C03628=1105.087,205.699,431.695,178.828,14.143,151.207
C03629=1105.092,205.948,431.670,178.832,14.142,151.206
C03630=1105.098,206.197,431.646,178.836,14.141,151.205
C03631=1105.103,206.446,431.621,178.840,14.139,151.203
C03632=1105.109,206.694,431.597,178.845,14.138,151.202
C03633=1105.115,206.943,431.573,178.848,14.136,151.201
C03634=1105.121,207.191,431.548,178.853,14.136,151.200
C03635=1105.126,207.440,431.524,178.857,14.134,151.198
C03636=1105.132,207.689,431.499,178.861,14.133,151.197
C03637=1105.156,208.685,431.402,178.887,14.133,151.191
C03638=1105.163,209.052,431.365,178.893,14.132,151.190
C03639=1105.171,209.419,431.330,178.899,14.131,151.188
C03640=1105.181,209.786,431.293,178.904,14.131,151.187
C03641=1105.189,210.152,431.257,178.911,14.131,151.186
C03642=1105.195,210.402,431.232,178.914,14.129,151.185
C03643=1105.200,210.650,431.208,178.918,14.129,151.184
C03644=1105.206,210.899,431.183,178.922,14.129,151.183
C03645=1105.211,211.147,431.159,178.926,14.129,151.182
C03646=1105.217,211.397,431.134,178.930,14.128,151.181
C03647=1105.223,211.645,431.109,178.934,14.127,151.180
C03648=1105.228,211.893,431.085,178.938,14.127,151.179
C03649=1105.234,212.143,431.060,178.942,14.126,151.178
C03650=1105.240,212.390,431.035,178.946,14.126,151.177
C03651=1105.246,212.640,431.010,178.949,14.125,151.176
C03652=1105.251,212.888,430.986,178.953,14.125,151.175
C03653=1105.256,213.137,430.960,178.958,14.125,151.174
C03654=1105.262,213.386,430.936,178.961,14.125,151.173
C03655=1105.268,213.635,430.911,178.966,14.124,151.172
C03656=1105.273,213.883,430.886,178.969,14.123,151.171
C03657=1105.279,214.132,430.861,178.973,14.123,151.170
C03658=1105.285,214.381,430.836,178.977,14.123,151.169
C03659=1105.291,214.629,430.812,178.981,14.122,151.168
C03660=1105.296,214.879,430.786,178.985,14.122,151.167
C03661=1105.302,215.127,430.761,178.989,14.122,151.166
C03662=1105.308,215.376,430.737,178.993,14.121,151.165
C03663=1105.313,215.624,430.712,178.997,14.120,151.164
C03664=1105.319,215.873,430.687,179.001,14.120,151.163
C03665=1105.325,216.121,430.662,179.005,14.120,151.162
C03666=1105.330,216.371,430.637,179.009,14.119,151.161
C03667=1105.335,216.619,430.612,179.012,14.119,151.160
C03668=1105.341,216.868,430.587,179.017,14.118,151.159
C03669=1105.348,217.117,430.562,179.020,14.118,151.158
C03670=1105.352,217.365,430.536,179.025,14.118,151.157
C03671=1105.358,217.614,430.512,179.029,14.118,151.156
C03672=1105.364,217.862,430.487,179.033,14.117,151.155
C03673=1105.370,218.111,430.461,179.036,14.116,151.154
C03674=1105.375,218.361,430.436,179.040,14.116,151.153
C03675=1105.381,218.608,430.411,179.044,14.116,151.152
C03676=1105.387,218.857,430.386,179.048,14.115,151.151
C03677=1105.392,219.106,430.362,179.052,14.115,151.150
C03678=1105.398,219.355,430.336,179.056,14.115,151.149
C03679=1105.404,219.603,430.310,179.060,14.114,151.148
C03680=1105.409,219.852,430.286,179.064,14.114,151.147
C03681=1105.415,220.101,430.260,179.068,14.113,151.146
C03682=1105.421,220.350,430.235,179.072,14.113,151.145
C03683=1105.427,220.598,430.210,179.076,14.113,151.144
C03684=1105.433,220.847,430.185,179.080,14.112,151.143
C03685=1105.438,221.096,430.159,179.083,14.112,151.142
C03686=1105.444,221.344,430.134,179.087,14.111,151.141
C03687=1105.450,221.592,430.109,179.092,14.111,151.140
C03688=1105.455,221.841,430.083,179.096,14.111,151.139
C03689=1105.461,222.089,430.058,179.100,14.110,151.138
C03690=1105.470,222.460,430.020,179.105,14.110,151.137
C03691=1105.477,222.831,429.983,179.111,14.109,151.135
C03692=1105.486,223.201,429.944,179.117,14.108,151.134
C03693=1105.494,223.571,429.907,179.123,14.108,151.133
C03694=1105.501,223.820,429.881,179.127,14.108,151.132
C03695=1105.506,224.068,429.856,179.131,14.107,151.131
C03696=1105.512,224.316,429.831,179.134,14.107,151.130
C03697=1105.517,224.565,429.805,179.139,14.107,151.129
C03698=1105.523,224.814,429.779,179.143,14.107,151.128
C03699=1105.528,225.062,429.754,179.147,14.106,151.127
C03700=1105.534,225.311,429.728,179.151,14.106,151.126
C03701=1105.540,225.560,429.702,179.155,14.106,151.125
C03702=1105.545,225.808,429.677,179.159,14.106,151.124
C03703=1105.551,226.057,429.652,179.162,14.105,151.123
C03704=1105.556,226.306,429.626,179.166,14.104,151.122
C03705=1105.563,226.555,429.600,179.170,14.104,151.121
C03706=1105.568,226.804,429.574,179.174,14.104,151.120
C03707=1105.574,227.052,429.549,179.178,14.104,151.119
C03708=1105.579,227.301,429.523,179.182,14.103,151.118
C03709=1105.585,227.549,429.498,179.186,14.103,151.117
C03710=1105.591,227.798,429.472,179.191,14.103,151.116
C03711=1105.596,228.047,429.447,179.194,14.102,151.115
C03712=1105.602,228.295,429.421,179.198,14.102,151.114
C03713=1105.608,228.544,429.395,179.202,14.102,151.113
C03714=1105.614,228.792,429.369,179.206,14.102,151.112
C03715=1105.619,229.041,429.343,179.210,14.101,151.111
C03716=1105.625,229.290,429.317,179.214,14.101,151.110
C03717=1105.631,229.538,429.292,179.218,14.101,151.109
C03718=1105.636,229.787,429.266,179.222,14.101,151.108
C03719=1105.642,230.035,429.240,179.226,14.100,151.107
C03720=1105.648,230.284,429.215,179.229,14.100,151.107
C03721=1105.654,230.533,429.188,179.234,14.099,151.105
C03722=1105.659,230.782,429.162,179.237,14.099,151.105
C03723=1105.665,231.030,429.137,179.241,14.099,151.104
C03724=1105.670,231.278,429.111,179.246,14.099,151.103
C03725=1105.676,231.527,429.084,179.250,14.099,151.102
C03726=1105.682,231.776,429.058,179.254,14.098,151.101
C03727=1105.688,232.024,429.033,179.258,14.098,151.100
C03728=1105.693,232.273,429.006,179.262,14.098,151.099
C03729=1105.699,232.522,428.981,179.266,14.098,151.098
C03730=1105.704,232.771,428.955,179.269,14.097,151.097
C03731=1105.710,233.018,428.928,179.273,14.097,151.096
C03732=1105.716,233.267,428.903,179.277,14.097,151.095
C03733=1105.722,233.515,428.876,179.281,14.096,151.094
C03734=1105.727,233.764,428.850,179.285,14.096,151.093
C03735=1105.733,234.013,428.825,179.289,14.096,151.092
C03736=1105.738,234.262,428.798,179.293,14.096,151.091
C03737=1105.744,234.510,428.773,179.297,14.096,151.090
C03738=1105.750,234.759,428.746,179.301,14.096,151.089
C03739=1105.756,235.008,428.720,179.305,14.096,151.089
C03740=1105.762,235.256,428.693,179.309,14.095,151.087
C03741=1105.766,235.504,428.668,179.313,14.095,151.087
C03742=1105.775,235.867,428.629,179.319,14.094,151.085
C03743=1105.783,236.228,428.591,179.324,14.094,151.084
C03744=1105.791,236.590,428.552,179.330,14.094,151.083
C03745=1105.799,236.952,428.514,179.336,14.094,151.081
C03746=1105.805,237.201,428.488,179.340,14.094,151.080
C03747=1105.810,237.449,428.461,179.344,14.093,151.079
C03748=1105.816,237.698,428.436,179.348,14.093,151.078
C03749=1105.822,237.946,428.409,179.351,14.093,151.077
C03750=1105.828,238.194,428.383,179.355,14.092,151.076
C03751=1105.834,238.443,428.357,179.359,14.092,151.075
C03752=1105.839,238.692,428.330,179.363,14.092,151.075
C03753=1105.845,238.940,428.304,179.367,14.092,151.074
C03754=1105.851,239.189,428.278,179.371,14.092,151.073
C03755=1105.856,239.437,428.251,179.375,14.092,151.072
C03756=1105.862,239.686,428.224,179.379,14.091,151.071
C03757=1105.868,239.935,428.198,179.383,14.091,151.070
C03758=1105.874,240.183,428.172,179.387,14.091,151.069
C03759=1105.879,240.432,428.145,179.391,14.091,151.068
C03760=1105.884,240.680,428.118,179.395,14.091,151.067
C03761=1105.890,240.929,428.092,179.399,14.091,151.066
C03762=1105.896,241.178,428.065,179.403,14.091,151.065
C03763=1105.902,241.426,428.038,179.407,14.090,151.064
C03764=1105.908,241.675,428.012,179.411,14.090,151.063
C03765=1105.913,241.923,427.985,179.415,14.090,151.062
C03766=1105.919,242.172,427.958,179.419,14.090,151.061
C03767=1105.925,242.420,427.932,179.423,14.090,151.060
C03768=1105.931,242.669,427.906,179.427,14.090,151.060
C03769=1105.936,242.917,427.879,179.431,14.090,151.059
C03770=1105.942,243.166,427.853,179.435,14.090,151.058
C03771=1105.947,243.414,427.825,179.439,14.090,151.057
C03772=1105.953,243.663,427.799,179.443,14.090,151.056
C03773=1105.959,243.911,427.772,179.446,14.089,151.055
C03774=1105.964,244.159,427.745,179.450,14.089,151.054
C03775=1105.970,244.409,427.718,179.454,14.089,151.053
C03776=1105.976,244.657,427.691,179.458,14.089,151.052
C03777=1105.982,244.905,427.664,179.462,14.089,151.051
C03778=1105.987,245.154,427.638,179.466,14.089,151.050
C03779=1105.992,245.402,427.611,179.470,14.088,151.049
C03780=1105.998,245.651,427.584,179.474,14.088,151.049
C03781=1106.004,245.899,427.557,179.478,14.088,151.048
C03782=1106.010,246.148,427.531,179.482,14.088,151.047
C03783=1106.015,246.396,427.503,179.486,14.088,151.046
C03784=1106.021,246.645,427.476,179.490,14.088,151.045
C03785=1106.027,246.894,427.450,179.494,14.088,151.044
C03786=1106.032,247.142,427.422,179.498,14.088,151.043
C03787=1106.038,247.391,427.396,179.501,14.088,151.042
C03788=1106.043,247.639,427.369,179.505,14.088,151.041
C03789=1106.049,247.888,427.342,179.510,14.087,151.040
C03790=1106.055,248.135,427.315,179.513,14.087,151.039
C03791=1106.060,248.384,427.288,179.517,14.087,151.039
C03792=1106.066,248.633,427.260,179.521,14.087,151.038
C03793=1106.072,248.882,427.234,179.525,14.087,151.037
C03794=1106.079,249.237,427.195,179.531,14.088,151.036
C03795=1106.087,249.591,427.156,179.537,14.087,151.034
C03796=1106.095,249.947,427.117,179.542,14.087,151.033
C03797=1106.104,250.302,427.079,179.548,14.088,151.032
C03798=1106.109,250.550,427.051,179.552,14.088,151.031
C03799=1106.115,250.799,427.024,179.556,14.088,151.030
C03800=1106.120,251.047,426.997,179.560,14.088,151.029
C03801=1106.127,251.296,426.969,179.564,14.088,151.028
C03802=1106.132,251.544,426.942,179.568,14.088,151.027
C03803=1106.137,251.793,426.915,179.572,14.088,151.026
C03804=1106.143,252.041,426.888,179.576,14.088,151.025
C03805=1106.149,252.290,426.861,179.579,14.088,151.025
C03806=1106.154,252.539,426.833,179.583,14.088,151.024
C03807=1106.159,252.787,426.805,179.587,14.088,151.023
C03808=1106.165,253.035,426.779,179.591,14.088,151.022
C03809=1106.170,253.284,426.751,179.595,14.088,151.021
C03810=1106.177,253.532,426.724,179.599,14.088,151.020
C03811=1106.182,253.781,426.696,179.603,14.088,151.019
C03812=1106.188,254.028,426.669,179.607,14.088,151.018
C03813=1106.194,254.278,426.641,179.611,14.088,151.018
C03814=1106.200,254.526,426.614,179.614,14.088,151.017
C03815=1106.205,254.774,426.587,179.619,14.087,151.016
C03816=1106.210,255.022,426.559,179.623,14.088,151.015
C03817=1106.217,255.271,426.532,179.627,14.088,151.014
C03818=1106.222,255.519,426.504,179.631,14.088,151.013
C03819=1106.228,255.768,426.477,179.635,14.088,151.012
C03820=1106.234,256.017,426.449,179.639,14.088,151.011
C03821=1106.239,256.265,426.422,179.643,14.088,151.010
C03822=1106.245,256.513,426.394,179.647,14.088,151.009
C03823=1106.251,256.762,426.366,179.650,14.088,151.009
C03824=1106.256,257.010,426.339,179.654,14.088,151.008
C03825=1106.262,257.258,426.311,179.658,14.088,151.007
C03826=1106.267,257.507,426.284,179.662,14.088,151.006
C03827=1106.273,257.756,426.256,179.666,14.088,151.005
C03828=1106.279,258.003,426.228,179.670,14.088,151.004
C03829=1106.284,258.253,426.201,179.674,14.088,151.003
C03830=1106.290,258.501,426.173,179.678,14.089,151.003
C03831=1106.296,258.749,426.145,179.681,14.089,151.002
C03832=1106.302,258.997,426.117,179.685,14.089,151.001
C03833=1106.307,259.246,426.090,179.690,14.089,151.000
C03834=1106.314,259.494,426.062,179.694,14.089,150.999
C03835=1106.319,259.742,426.034,179.698,14.089,150.998
C03836=1106.325,259.991,426.006,179.702,14.089,150.997
C03837=1106.331,260.239,425.979,179.706,14.089,150.996
C03838=1106.336,260.487,425.951,179.710,14.089,150.995
C03839=1106.342,260.736,425.923,179.714,14.089,150.995
C03840=1106.347,260.984,425.895,179.717,14.089,150.994
C03841=1106.354,261.233,425.867,179.721,14.089,150.993
C03842=1106.359,261.481,425.840,179.725,14.089,150.992
C03843=1106.365,261.730,425.812,179.729,14.089,150.991
C03844=1106.370,261.978,425.784,179.733,14.089,150.990
C03845=1106.377,262.227,425.756,179.737,14.089,150.989
C03846=1106.385,262.579,425.716,179.743,14.090,150.988
C03847=1106.393,262.931,425.676,179.748,14.090,150.987
C03848=1106.400,263.284,425.637,179.754,14.091,150.986
C03849=1106.409,263.636,425.597,179.759,14.090,150.984
C03850=1106.414,263.885,425.569,179.763,14.090,150.984
C03851=1106.421,264.133,425.541,179.767,14.091,150.983
C03852=1106.426,264.381,425.513,179.771,14.091,150.982
C03853=1106.432,264.630,425.485,179.775,14.091,150.981
C03854=1106.438,264.878,425.457,179.779,14.091,150.980
C03855=1106.444,265.127,425.429,179.783,14.091,150.979
C03856=1106.449,265.375,425.401,179.787,14.092,150.979
C03857=1106.455,265.623,425.373,179.791,14.092,150.978
C03858=1106.460,265.871,425.345,179.795,14.092,150.977
C03859=1106.466,266.120,425.316,179.798,14.092,150.976
C03860=1106.472,266.368,425.288,179.802,14.092,150.975
C03861=1106.478,266.616,425.259,179.806,14.092,150.974
C03862=1106.483,266.864,425.231,179.810,14.093,150.973
C03863=1106.489,267.113,425.203,179.814,14.093,150.973
C03864=1106.494,267.361,425.175,179.818,14.093,150.972
C03865=1106.500,267.610,425.147,179.822,14.093,150.971
C03866=1106.506,267.857,425.118,179.826,14.093,150.970
C03867=1106.512,268.106,425.090,179.830,14.094,150.969
C03868=1106.517,268.354,425.062,179.833,14.094,150.968
C03869=1106.523,268.603,425.033,179.837,14.094,150.968
C03870=1106.529,268.852,425.005,179.842,14.095,150.967
C03871=1106.535,269.099,424.976,179.846,14.095,150.966
C03872=1106.540,269.348,424.947,179.850,14.095,150.965
C03873=1106.545,269.596,424.920,179.853,14.095,150.964
C03874=1106.551,269.845,424.891,179.857,14.095,150.963
C03875=1106.557,270.092,424.863,179.861,14.095,150.963
C03876=1106.563,270.341,424.834,179.865,14.096,150.962
C03877=1106.569,270.590,424.806,179.869,14.097,150.961
C03878=1106.574,270.837,424.777,179.873,14.097,150.960
C03879=1106.580,271.086,424.748,179.877,14.097,150.959
C03880=1106.585,271.334,424.720,179.881,14.097,150.958
C03881=1106.591,271.583,424.691,179.884,14.097,150.958
C03882=1106.597,271.831,424.663,179.888,14.097,150.957
C03883=1106.603,272.079,424.634,179.892,14.097,150.956
C03884=1106.608,272.328,424.605,179.896,14.099,150.955
C03885=1106.613,272.576,424.577,179.900,14.099,150.954
C03886=1106.620,272.824,424.548,179.904,14.099,150.954
C03887=1106.626,273.073,424.520,179.907,14.099,150.953
C03888=1106.631,273.320,424.491,179.911,14.099,150.952
C03889=1106.636,273.569,424.462,179.915,14.099,150.951
C03890=1106.643,273.817,424.433,179.920,14.100,150.950
C03891=1106.648,274.065,424.405,179.923,14.101,150.950
C03892=1106.654,274.314,424.376,179.927,14.101,150.949
C03893=1106.659,274.562,424.348,179.931,14.101,150.948
C03894=1106.665,274.810,424.319,179.935,14.101,150.947
C03895=1106.671,275.059,424.290,179.939,14.102,150.946
C03896=1106.676,275.307,424.261,179.943,14.102,150.946
C03897=1106.682,275.555,424.232,179.947,14.103,150.945
C03898=1106.690,275.910,424.191,179.952,14.102,150.944
C03899=1106.698,276.266,424.149,179.957,14.104,150.943
C03900=1106.707,276.621,424.109,179.963,14.104,150.941
C03901=1106.715,276.976,424.067,179.968,14.105,150.940
C03902=1106.720,277.224,424.038,179.972,14.105,150.939
C03903=1106.726,277.473,424.010,179.977,14.106,150.939
C03904=1106.732,277.721,423.980,179.980,14.106,150.938
C03905=1106.737,277.970,423.951,179.984,14.106,150.937
C03906=1106.743,278.217,423.922,179.988,14.106,150.936
C03907=1106.748,278.466,423.893,179.992,14.107,150.936
C03908=1106.755,278.714,423.864,179.996,14.108,150.935
C03909=1106.759,278.962,423.835,180.000,14.108,150.934
C03910=1106.766,279.210,423.806,-179.997,14.108,150.933
C03911=1106.771,279.459,423.777,-179.993,14.108,150.932
C03912=1106.777,279.707,423.748,-179.989,14.109,150.932
C03913=1106.782,279.955,423.719,-179.985,14.110,150.931
C03914=1106.788,280.203,423.690,-179.981,14.110,150.930
C03915=1106.794,280.452,423.660,-179.977,14.110,150.929
C03916=1106.800,280.700,423.631,-179.974,14.111,150.929
C03917=1106.806,280.948,423.601,-179.969,14.111,150.928
C03918=1106.811,281.196,423.573,-179.966,14.112,150.927
C03919=1106.816,281.445,423.544,-179.962,14.112,150.926
C03920=1106.823,281.693,423.515,-179.958,14.112,150.926
C03921=1106.828,281.941,423.485,-179.955,14.113,150.925
C03922=1106.834,282.189,423.456,-179.950,14.114,150.924
C03923=1106.839,282.437,423.427,-179.947,14.114,150.923
C03924=1106.845,282.685,423.397,-179.943,14.114,150.923
C03925=1106.851,282.934,423.368,-179.939,14.115,150.922
C03926=1106.856,283.181,423.339,-179.935,14.116,150.921
C03927=1106.862,283.430,423.309,-179.931,14.116,150.920
C03928=1106.868,283.678,423.280,-179.928,14.117,150.920
C03929=1106.873,283.926,423.250,-179.924,14.117,150.919
C03930=1106.879,284.175,423.221,-179.919,14.118,150.918
C03931=1106.885,284.423,423.192,-179.916,14.118,150.917
C03932=1106.890,284.671,423.163,-179.912,14.118,150.917
C03933=1106.896,284.919,423.133,-179.909,14.119,150.916
C03934=1106.902,285.167,423.104,-179.904,14.120,150.915
C03935=1106.908,285.415,423.074,-179.900,14.120,150.914
C03936=1106.913,285.664,423.044,-179.897,14.121,150.914
C03937=1106.919,285.912,423.014,-179.893,14.122,150.913
C03938=1106.924,286.159,422.986,-179.889,14.122,150.912
C03939=1106.930,286.408,422.956,-179.885,14.122,150.911
C03940=1106.935,286.656,422.926,-179.882,14.123,150.911
C03941=1106.942,286.904,422.897,-179.878,14.124,150.910
C03942=1106.947,287.152,422.867,-179.874,14.124,150.909
C03943=1106.953,287.401,422.837,-179.870,14.125,150.909
C03944=1106.958,287.649,422.808,-179.867,14.125,150.908
C03945=1106.965,287.897,422.779,-179.862,14.126,150.907
C03946=1106.970,288.145,422.748,-179.859,14.126,150.906
C03947=1106.975,288.393,422.719,-179.855,14.127,150.906
C03948=1106.981,288.641,422.689,-179.850,14.128,150.905
C03949=1106.987,288.889,422.659,-179.847,14.128,150.904
C03950=1106.996,289.254,422.616,-179.841,14.129,150.903
C03951=1107.005,289.619,422.572,-179.836,14.130,150.902
C03952=1107.013,289.983,422.528,-179.830,14.130,150.901
C03953=1107.020,290.348,422.484,-179.825,14.132,150.900
C03954=1107.027,290.596,422.455,-179.821,14.132,150.899
C03955=1107.032,290.845,422.425,-179.817,14.133,150.899
C03956=1107.038,291.093,422.395,-179.813,14.134,150.898
C03957=1107.043,291.341,422.365,-179.810,14.134,150.897
C03958=1107.049,291.589,422.335,-179.806,14.135,150.896
C03959=1107.055,291.837,422.305,-179.802,14.136,150.896
C03960=1107.061,292.085,422.275,-179.798,14.136,150.895
C03961=1107.066,292.334,422.245,-179.794,14.137,150.894
C03962=1107.072,292.581,422.215,-179.791,14.138,150.894
C03963=1107.077,292.830,422.185,-179.787,14.138,150.893
C03964=1107.083,293.078,422.155,-179.783,14.139,150.892
C03965=1107.089,293.326,422.125,-179.779,14.140,150.892
C03966=1107.095,293.574,422.095,-179.776,14.140,150.891
C03967=1107.100,293.822,422.065,-179.771,14.142,150.890
C03968=1107.106,294.070,422.035,-179.768,14.142,150.890
C03969=1107.112,294.318,422.005,-179.764,14.143,150.889
C03970=1107.117,294.567,421.975,-179.760,14.144,150.888
C03971=1107.123,294.814,421.945,-179.756,14.144,150.887
C03972=1107.129,295.062,421.914,-179.753,14.145,150.887
C03973=1107.134,295.311,421.885,-179.749,14.146,150.886
C03974=1107.140,295.558,421.854,-179.745,14.146,150.885
C03975=1107.146,295.806,421.824,-179.742,14.147,150.885
C03976=1107.152,296.055,421.794,-179.737,14.148,150.884
C03977=1107.157,296.303,421.764,-179.734,14.148,150.883
C03978=1107.162,296.551,421.733,-179.730,14.149,150.883
C03979=1107.168,296.799,421.703,-179.726,14.150,150.882
C03980=1107.174,297.047,421.673,-179.723,14.151,150.881
C03981=1107.180,297.295,421.643,-179.719,14.152,150.881
C03982=1107.185,297.543,421.612,-179.715,14.153,150.880
C03983=1107.191,297.790,421.582,-179.712,14.153,150.879
C03984=1107.197,298.039,421.552,-179.707,14.155,150.879
C03985=1107.202,298.287,421.521,-179.704,14.155,150.878
C03986=1107.208,298.535,421.491,-179.700,14.156,150.877
C03987=1107.214,298.783,421.460,-179.696,14.157,150.877
C03988=1107.220,299.031,421.430,-179.693,14.157,150.876
C03989=1107.225,299.280,421.400,-179.689,14.159,150.876
C03990=1107.230,299.528,421.369,-179.685,14.159,150.875
C03991=1107.236,299.776,421.339,-179.682,14.160,150.874
C03992=1107.241,300.024,421.308,-179.677,14.161,150.874
C03993=1107.247,300.271,421.278,-179.674,14.162,150.873
C03994=1107.253,300.519,421.247,-179.670,14.163,150.872
C03995=1107.258,300.767,421.216,-179.666,14.164,150.872
C03996=1107.264,301.015,421.186,-179.663,14.164,150.871
C03997=1107.270,301.263,421.156,-179.659,14.166,150.871
C03998=1107.275,301.511,421.125,-179.656,14.166,150.870
C03999=1107.281,301.759,421.094,-179.651,14.168,150.869
C04000=1107.286,302.007,421.063,-179.648,14.168,150.869
C04001=1107.292,302.256,421.033,-179.645,14.169,150.868
C04002=1107.300,302.634,420.987,-179.638,14.171,150.867
C04003=1107.309,303.013,420.939,-179.633,14.172,150.866
C04004=1107.318,303.391,420.892,-179.627,14.174,150.865
C04005=1107.326,303.770,420.846,-179.622,14.175,150.864
C04006=1107.331,304.018,420.815,-179.618,14.176,150.864
C04007=1107.337,304.266,420.785,-179.614,14.177,150.863
C04008=1107.343,304.514,420.753,-179.610,14.178,150.862
C04009=1107.349,304.762,420.722,-179.607,14.179,150.862
C04010=1107.355,305.010,420.692,-179.603,14.180,150.861
C04011=1107.360,305.258,420.661,-179.599,14.181,150.861
C04012=1107.366,305.506,420.631,-179.595,14.182,150.860
C04013=1107.372,305.754,420.598,-179.592,14.183,150.859
C04014=1107.378,306.002,420.568,-179.589,14.184,150.859
C04015=1107.383,306.250,420.537,-179.584,14.185,150.858
C04016=1107.389,306.498,420.507,-179.581,14.185,150.858
C04017=1107.394,306.745,420.475,-179.577,14.187,150.857
C04018=1107.400,306.994,420.444,-179.573,14.188,150.856
C04019=1107.405,307.242,420.414,-179.570,14.189,150.856
C04020=1107.412,307.489,420.382,-179.566,14.190,150.855
C04021=1107.417,307.737,420.352,-179.562,14.191,150.855
C04022=1107.423,307.986,420.321,-179.559,14.192,150.854
C04023=1107.428,308.233,420.289,-179.555,14.194,150.854
C04024=1107.433,308.482,420.258,-179.551,14.194,150.853
C04025=1107.440,308.730,420.227,-179.547,14.195,150.852
C04026=1107.445,308.978,420.196,-179.544,14.196,150.852
C04027=1107.451,309.225,420.165,-179.540,14.197,150.851
C04028=1107.457,309.474,420.133,-179.536,14.198,150.851
C04029=1107.463,309.721,420.103,-179.533,14.199,150.850
C04030=1107.468,309.970,420.072,-179.529,14.201,150.849
C04031=1107.474,310.218,420.040,-179.526,14.201,150.849
C04032=1107.480,310.466,420.010,-179.522,14.203,150.848
C04033=1107.485,310.713,419.978,-179.518,14.204,150.848
C04034=1107.492,310.962,419.947,-179.514,14.205,150.847
C04035=1107.497,311.209,419.916,-179.511,14.206,150.847
C04036=1107.502,311.457,419.885,-179.507,14.207,150.846
C04037=1107.509,311.705,419.853,-179.504,14.208,150.845
C04038=1107.514,311.953,419.822,-179.499,14.209,150.845
C04039=1107.520,312.202,419.790,-179.496,14.210,150.844
C04040=1107.526,312.449,419.759,-179.492,14.212,150.844
C04041=1107.531,312.697,419.728,-179.489,14.212,150.843
C04042=1107.537,312.945,419.696,-179.485,14.214,150.843
C04043=1107.543,313.192,419.665,-179.481,14.214,150.842
C04044=1107.549,313.441,419.634,-179.478,14.216,150.842
C04045=1107.554,313.689,419.602,-179.474,14.217,150.841
C04046=1107.561,313.937,419.571,-179.470,14.218,150.840
C04047=1107.566,314.185,419.540,-179.467,14.219,150.840
C04048=1107.571,314.432,419.508,-179.463,14.221,150.839
C04049=1107.577,314.680,419.476,-179.460,14.221,150.839
C04050=1107.583,314.928,419.446,-179.456,14.223,150.838
C04051=1107.589,315.176,419.414,-179.453,14.224,150.838
C04052=1107.595,315.424,419.382,-179.449,14.226,150.837
C04053=1107.601,315.672,419.350,-179.445,14.226,150.837
C04054=1107.609,316.053,419.302,-179.440,14.229,150.836
C04055=1107.617,316.434,419.253,-179.434,14.230,150.835
C04056=1107.626,316.816,419.205,-179.428,14.233,150.834
C04057=1107.634,317.197,419.156,-179.423,14.234,150.834
C04058=1107.640,317.445,419.125,-179.419,14.236,150.833
C04059=1107.646,317.693,419.093,-179.416,14.237,150.833
C04060=1107.651,317.941,419.061,-179.412,14.239,150.832
C04061=1107.657,318.189,419.029,-179.409,14.240,150.832
C04062=1107.662,318.436,418.997,-179.405,14.241,150.831
C04063=1107.668,318.685,418.965,-179.401,14.243,150.831
C04064=1107.674,318.932,418.934,-179.398,14.244,150.830
C04065=1107.680,319.181,418.902,-179.394,14.245,150.830
C04066=1107.685,319.428,418.871,-179.391,14.246,150.829
C04067=1107.691,319.677,418.839,-179.387,14.248,150.829
C04068=1107.696,319.924,418.807,-179.383,14.250,150.828
C04069=1107.702,320.172,418.775,-179.380,14.251,150.828
C04070=1107.708,320.420,418.743,-179.376,14.252,150.827
C04071=1107.714,320.668,418.711,-179.374,14.254,150.827
C04072=1107.718,320.916,418.679,-179.370,14.255,150.827
C04073=1107.724,321.164,418.647,-179.367,14.256,150.826
C04074=1107.730,321.412,418.615,-179.363,14.258,150.826
C04075=1107.736,321.659,418.582,-179.359,14.259,150.825
C04076=1107.741,321.907,418.551,-179.356,14.260,150.825
C04077=1107.747,322.155,418.519,-179.352,14.262,150.824
C04078=1107.753,322.403,418.487,-179.349,14.263,150.824
C04079=1107.759,322.651,418.455,-179.345,14.265,150.823
C04080=1107.764,322.899,418.422,-179.341,14.267,150.823
C04081=1107.769,323.147,418.391,-179.338,14.268,150.822
C04082=1107.775,323.395,418.359,-179.334,14.269,150.822
C04083=1107.781,323.642,418.326,-179.331,14.271,150.822
C04084=1107.787,323.890,418.294,-179.327,14.272,150.821
C04085=1107.793,324.138,418.262,-179.324,14.274,150.821
C04086=1107.798,324.386,418.230,-179.320,14.275,150.820
C04087=1107.804,324.634,418.198,-179.317,14.277,150.820
C04088=1107.810,324.882,418.165,-179.313,14.278,150.819
C04089=1107.815,325.129,418.134,-179.310,14.279,150.819
C04090=1107.821,325.378,418.101,-179.306,14.281,150.818
C04091=1107.826,325.626,418.069,-179.302,14.283,150.818
C04092=1107.832,325.873,418.037,-179.299,14.284,150.818
C04093=1107.838,326.121,418.005,-179.295,14.286,150.817
C04094=1107.844,326.369,417.973,-179.292,14.288,150.817
C04095=1107.849,326.617,417.940,-179.289,14.289,150.816
C04096=1107.855,326.865,417.908,-179.285,14.290,150.816
C04097=1107.861,327.113,417.876,-179.282,14.292,150.816
C04098=1107.866,327.360,417.843,-179.278,14.293,150.815
C04099=1107.872,327.609,417.811,-179.274,14.295,150.815
C04100=1107.878,327.856,417.778,-179.271,14.296,150.814
C04101=1107.884,328.104,417.746,-179.267,14.298,150.814
C04102=1107.889,328.352,417.713,-179.264,14.300,150.814
C04103=1107.895,328.600,417.681,-179.261,14.301,150.813
C04104=1107.901,328.848,417.649,-179.257,14.303,150.813
C04105=1107.906,329.095,417.616,-179.253,14.304,150.812
C04106=1107.915,329.470,417.566,-179.248,14.306,150.812
C04107=1107.923,329.844,417.518,-179.243,14.309,150.811
C04108=1107.932,330.218,417.468,-179.237,14.312,150.811
C04109=1107.942,330.592,417.419,-179.233,14.314,150.810
C04110=1107.947,330.840,417.387,-179.229,14.316,150.810
C04111=1107.953,331.088,417.355,-179.225,14.318,150.809
C04112=1107.959,331.336,417.321,-179.222,14.319,150.809
C04113=1107.964,331.584,417.289,-179.218,14.321,150.808
C04114=1107.971,331.831,417.256,-179.215,14.323,150.808
C04115=1107.976,332.079,417.223,-179.212,14.324,150.808
C04116=1107.982,332.327,417.191,-179.208,14.326,150.807
C04117=1107.987,332.575,417.158,-179.205,14.328,150.807
C04118=1107.994,332.822,417.125,-179.201,14.330,150.807
C04119=1107.999,333.071,417.093,-179.198,14.331,150.806
C04120=1108.004,333.318,417.060,-179.194,14.333,150.806
C04121=1108.010,333.566,417.027,-179.191,14.335,150.806
C04122=1108.016,333.814,416.994,-179.187,14.337,150.805
C04123=1108.022,334.062,416.962,-179.184,14.338,150.805
C04124=1108.027,334.310,416.928,-179.181,14.340,150.805
C04125=1108.032,334.557,416.895,-179.177,14.342,150.804
C04126=1108.038,334.805,416.863,-179.174,14.344,150.804
C04127=1108.044,335.052,416.829,-179.171,14.345,150.804
C04128=1108.050,335.301,416.797,-179.167,14.347,150.803
C04129=1108.056,335.549,416.764,-179.164,14.349,150.803
C04130=1108.060,335.796,416.731,-179.160,14.351,150.803
C04131=1108.067,336.043,416.698,-179.157,14.352,150.802
C04132=1108.072,336.291,416.665,-179.153,14.354,150.802
C04133=1108.078,336.539,416.631,-179.150,14.357,150.802
C04134=1108.084,336.787,416.599,-179.146,14.359,150.801
C04135=1108.089,337.035,416.566,-179.143,14.361,150.801
C04136=1108.095,337.283,416.533,-179.140,14.362,150.801
C04137=1108.101,337.531,416.500,-179.136,14.364,150.801
C04138=1108.106,337.778,416.467,-179.133,14.366,150.800
C04139=1108.112,338.026,416.434,-179.129,14.368,150.800
C04140=1108.117,338.274,416.400,-179.126,14.370,150.800
C04141=1108.124,338.521,416.368,-179.123,14.371,150.799
C04142=1108.129,338.769,416.334,-179.120,14.373,150.799
C04143=1108.135,339.017,416.301,-179.116,14.376,150.799
C04144=1108.140,339.265,416.268,-179.113,14.378,150.799
C04145=1108.147,339.512,416.234,-179.109,14.380,150.798
C04146=1108.152,339.760,416.201,-179.106,14.382,150.798
C04147=1108.158,340.008,416.167,-179.103,14.383,150.798
C04148=1108.163,340.255,416.135,-179.099,14.385,150.797
C04149=1108.168,340.503,416.101,-179.096,14.388,150.797
C04150=1108.174,340.751,416.068,-179.093,14.390,150.797
C04151=1108.180,340.999,416.035,-179.089,14.392,150.797
C04152=1108.186,341.246,416.002,-179.086,14.394,150.796
C04153=1108.191,341.494,415.968,-179.082,14.396,150.796
C04154=1108.197,341.742,415.934,-179.080,14.398,150.796
C04155=1108.203,341.989,415.901,-179.076,14.400,150.796
C04156=1108.208,342.237,415.868,-179.073,14.402,150.796
C04157=1108.214,342.485,415.834,-179.069,14.404,150.795
C04158=1108.223,342.853,415.785,-179.064,14.408,150.795
C04159=1108.231,343.221,415.735,-179.059,14.411,150.795
C04160=1108.240,343.589,415.685,-179.055,14.414,150.794
C04161=1108.248,343.957,415.636,-179.049,14.417,150.794
C04162=1108.254,344.205,415.601,-179.046,14.419,150.794
C04163=1108.259,344.453,415.568,-179.043,14.421,150.793
C04164=1108.265,344.700,415.535,-179.040,14.424,150.793
C04165=1108.271,344.948,415.501,-179.036,14.426,150.793
C04166=1108.276,345.196,415.467,-179.033,14.428,150.793
C04167=1108.282,345.443,415.433,-179.029,14.430,150.793
C04168=1108.288,345.691,415.400,-179.026,14.432,150.793
C04169=1108.293,345.939,415.367,-179.023,14.434,150.792
C04170=1108.299,346.186,415.333,-179.020,14.436,150.792
C04171=1108.305,346.434,415.299,-179.017,14.439,150.792
C04172=1108.311,346.681,415.265,-179.013,14.441,150.792
C04173=1108.316,346.929,415.232,-179.010,14.443,150.792
C04174=1108.321,347.177,415.197,-179.007,14.446,150.791
C04175=1108.327,347.425,415.164,-179.003,14.448,150.791
C04176=1108.333,347.672,415.130,-179.000,14.450,150.791
C04177=1108.338,347.920,415.096,-178.997,14.452,150.791
C04178=1108.345,348.168,415.062,-178.994,14.455,150.791
C04179=1108.350,348.416,415.029,-178.990,14.457,150.791
C04180=1108.356,348.663,414.995,-178.987,14.459,150.790
C04181=1108.361,348.911,414.960,-178.984,14.462,150.790
C04182=1108.367,349.158,414.927,-178.981,14.464,150.790
C04183=1108.373,349.406,414.893,-178.978,14.467,150.790
C04184=1108.378,349.653,414.859,-178.974,14.469,150.790
C04185=1108.384,349.901,414.825,-178.971,14.471,150.790
C04186=1108.390,350.148,414.791,-178.968,14.474,150.790
C04187=1108.395,350.396,414.757,-178.964,14.476,150.789
C04188=1108.401,350.644,414.723,-178.961,14.478,150.789
C04189=1108.406,350.891,414.689,-178.958,14.481,150.789
C04190=1108.413,351.139,414.655,-178.955,14.483,150.789
C04191=1108.418,351.387,414.621,-178.952,14.486,150.789
C04192=1108.424,351.634,414.587,-178.948,14.488,150.789
C04193=1108.429,351.882,414.553,-178.945,14.491,150.789
C04194=1108.435,352.129,414.519,-178.942,14.493,150.789
C04195=1108.440,352.377,414.484,-178.939,14.495,150.789
C04196=1108.446,352.625,414.451,-178.936,14.498,150.788
C04197=1108.452,352.873,414.416,-178.932,14.500,150.788
C04198=1108.458,353.120,414.382,-178.929,14.503,150.788
C04199=1108.463,353.367,414.348,-178.926,14.505,150.788
C04200=1108.469,353.615,414.314,-178.923,14.508,150.788
C04201=1108.474,353.862,414.279,-178.920,14.510,150.788
C04202=1108.480,354.110,414.245,-178.917,14.513,150.788
C04203=1108.486,354.358,414.211,-178.914,14.515,150.788
C04204=1108.492,354.606,414.176,-178.911,14.518,150.788
C04205=1108.497,354.853,414.142,-178.908,14.521,150.788
C04206=1108.503,355.101,414.108,-178.904,14.523,150.788
C04207=1108.508,355.348,414.074,-178.901,14.525,150.787
C04208=1108.513,355.596,414.039,-178.898,14.529,150.788
C04209=1108.520,355.844,414.005,-178.894,14.531,150.787
C04210=1108.528,356.213,413.954,-178.890,14.535,150.787
C04211=1108.538,356.583,413.901,-178.885,14.539,150.787
C04212=1108.545,356.954,413.850,-178.881,14.543,150.787
C04213=1108.554,357.323,413.799,-178.876,14.547,150.787
C04214=1108.559,357.572,413.764,-178.873,14.550,150.787
C04215=1108.565,357.819,413.730,-178.870,14.552,150.787
C04216=1108.570,358.067,413.695,-178.867,14.555,150.787
C04217=1108.576,358.314,413.661,-178.863,14.558,150.787
C04218=1108.582,358.562,413.625,-178.860,14.561,150.787
C04219=1108.588,358.809,413.591,-178.857,14.564,150.787
C04220=1108.593,359.057,413.556,-178.854,14.566,150.787
C04221=1108.599,359.304,413.522,-178.851,14.569,150.787
C04222=1108.605,359.552,413.487,-178.849,14.572,150.787
C04223=1108.611,359.799,413.453,-178.845,14.574,150.787
C04224=1108.616,360.046,413.418,-178.842,14.577,150.787
C04225=1108.622,360.294,413.384,-178.839,14.580,150.787
C04226=1108.628,360.541,413.348,-178.836,14.583,150.787
C04227=1108.633,360.789,413.314,-178.833,14.586,150.787
C04228=1108.639,361.036,413.280,-178.830,14.588,150.787
C04229=1108.645,361.284,413.244,-178.827,14.591,150.787
C04230=1108.650,361.531,413.209,-178.824,14.594,150.787
C04231=1108.656,361.779,413.175,-178.821,14.596,150.787
C04232=1108.662,362.026,413.139,-178.817,14.600,150.787
C04233=1108.667,362.274,413.105,-178.815,14.603,150.787
C04234=1108.673,362.521,413.071,-178.812,14.606,150.787
C04235=1108.679,362.769,413.035,-178.809,14.608,150.787
C04236=1108.684,363.017,413.000,-178.806,14.611,150.787
C04237=1108.689,363.264,412.965,-178.802,14.615,150.788
C04238=1108.696,363.512,412.930,-178.800,14.618,150.788
C04239=1108.701,363.758,412.895,-178.797,14.620,150.788
C04240=1108.706,364.006,412.860,-178.794,14.623,150.788
C04241=1108.713,364.253,412.825,-178.791,14.626,150.788
C04242=1108.718,364.501,412.791,-178.787,14.630,150.788
C04243=1108.724,364.748,412.755,-178.785,14.632,150.788
C04244=1108.730,364.996,412.720,-178.782,14.635,150.788
C04245=1108.735,365.243,412.685,-178.779,14.638,150.788
C04246=1108.741,365.491,412.651,-178.776,14.641,150.788
C04247=1108.747,365.738,412.615,-178.773,14.645,150.788
C04248=1108.752,365.986,412.581,-178.770,14.647,150.788
C04249=1108.758,366.234,412.545,-178.767,14.650,150.789
C04250=1108.763,366.480,412.509,-178.765,14.653,150.789
C04251=1108.769,366.728,412.475,-178.761,14.657,150.789
C04252=1108.775,366.975,412.440,-178.758,14.660,150.789
C04253=1108.781,367.222,412.404,-178.756,14.663,150.789
C04254=1108.786,367.470,412.370,-178.752,14.667,150.789
C04255=1108.792,367.718,412.334,-178.749,14.670,150.789
C04256=1108.797,367.965,412.299,-178.747,14.673,150.789
C04257=1108.803,368.212,412.263,-178.744,14.676,150.790
C04258=1108.808,368.460,412.228,-178.740,14.679,150.790
C04259=1108.814,368.707,412.193,-178.738,14.682,150.790
C04260=1108.820,368.955,412.157,-178.735,14.685,150.790
C04261=1108.825,369.202,412.122,-178.732,14.689,150.790
C04262=1108.834,369.587,412.067,-178.728,14.694,150.791
C04263=1108.843,369.972,412.011,-178.723,14.699,150.791
C04264=1108.852,370.356,411.957,-178.719,14.704,150.791
C04265=1108.861,370.742,411.902,-178.715,14.709,150.791
C04266=1108.866,370.989,411.866,-178.711,14.712,150.792
C04267=1108.872,371.236,411.831,-178.708,14.716,150.792
C04268=1108.878,371.483,411.795,-178.706,14.719,150.792
C04269=1108.884,371.731,411.759,-178.703,14.723,150.792
C04270=1108.889,371.978,411.724,-178.700,14.726,150.792
C04271=1108.895,372.225,411.688,-178.697,14.729,150.793
C04272=1108.900,372.473,411.652,-178.694,14.733,150.793
C04273=1108.906,372.720,411.617,-178.692,14.736,150.793
C04274=1108.911,372.967,411.581,-178.689,14.739,150.793
C04275=1108.917,373.215,411.546,-178.686,14.743,150.793
C04276=1108.923,373.462,411.510,-178.683,14.746,150.794
C04277=1108.929,373.710,411.474,-178.681,14.749,150.794
C04278=1108.934,373.957,411.439,-178.677,14.753,150.794
C04279=1108.940,374.204,411.403,-178.675,14.756,150.794
C04280=1108.946,374.451,411.368,-178.672,14.760,150.795
C04281=1108.952,374.699,411.332,-178.669,14.763,150.795
C04282=1108.956,374.946,411.296,-178.667,14.766,150.795
C04283=1108.963,375.193,411.260,-178.663,14.770,150.795
C04284=1108.968,375.440,411.225,-178.661,14.774,150.796
C04285=1108.974,375.688,411.189,-178.658,14.778,150.796
C04286=1108.979,375.935,411.153,-178.655,14.781,150.796
C04287=1108.985,376.183,411.117,-178.653,14.785,150.797
C04288=1108.991,376.430,411.081,-178.650,14.788,150.797
C04289=1108.997,376.677,411.045,-178.647,14.792,150.797
C04290=1109.002,376.925,411.009,-178.644,14.796,150.798
C04291=1109.007,377.172,410.974,-178.642,14.799,150.798
C04292=1109.014,377.419,410.937,-178.639,14.803,150.798
C04293=1109.018,377.666,410.901,-178.636,14.807,150.799
C04294=1109.024,377.914,410.865,-178.633,14.810,150.799
C04295=1109.030,378.160,410.829,-178.631,14.814,150.799
C04296=1109.035,378.408,410.793,-178.629,14.817,150.799
C04297=1109.041,378.656,410.757,-178.626,14.821,150.800
C04298=1109.047,378.902,410.721,-178.623,14.825,150.800
C04299=1109.053,379.150,410.685,-178.620,14.829,150.800
C04300=1109.058,379.397,410.650,-178.618,14.832,150.801
C04301=1109.064,379.644,410.613,-178.615,14.836,150.801
C04302=1109.070,379.892,410.577,-178.612,14.840,150.802
C04303=1109.075,380.139,410.541,-178.610,14.844,150.802
C04304=1109.081,380.386,410.505,-178.607,14.848,150.802
C04305=1109.086,380.633,410.468,-178.604,14.852,150.803
C04306=1109.092,380.881,410.433,-178.602,14.855,150.803
C04307=1109.098,381.128,410.396,-178.599,14.859,150.803
C04308=1109.103,381.375,410.360,-178.597,14.863,150.804
C04309=1109.110,381.622,410.324,-178.594,14.867,150.804
C04310=1109.115,381.870,410.287,-178.592,14.871,150.805
C04311=1109.121,382.116,410.251,-178.588,14.875,150.805
C04312=1109.126,382.364,410.215,-178.585,14.879,150.805
C04313=1109.132,382.611,410.179,-178.583,14.882,150.806
C04314=1109.141,383.022,410.118,-178.579,14.890,150.807
C04315=1109.151,383.434,410.058,-178.575,14.896,150.807
C04316=1109.160,383.846,409.997,-178.570,14.903,150.808
C04317=1109.170,384.258,409.936,-178.566,14.910,150.809
C04318=1109.175,384.504,409.900,-178.564,14.913,150.809
C04319=1109.180,384.752,409.863,-178.561,14.918,150.810
C04320=1109.187,384.999,409.827,-178.559,14.921,150.810
C04321=1109.192,385.246,409.790,-178.556,14.926,150.811
C04322=1109.197,385.493,409.753,-178.553,14.930,150.811
C04323=1109.204,385.740,409.717,-178.551,14.934,150.812
C04324=1109.208,385.988,409.681,-178.548,14.938,150.812
C04325=1109.215,386.235,409.644,-178.546,14.943,150.813
C04326=1109.220,386.482,409.607,-178.543,14.946,150.813
C04327=1109.225,386.729,409.571,-178.541,14.951,150.814
C04328=1109.232,386.976,409.534,-178.539,14.955,150.814
C04329=1109.237,387.224,409.498,-178.536,14.959,150.815
C04330=1109.242,387.471,409.461,-178.533,14.964,150.815
C04331=1109.248,387.717,409.425,-178.531,14.967,150.816
C04332=1109.254,387.965,409.388,-178.529,14.972,150.816
C04333=1109.259,388.212,409.351,-178.526,14.977,150.817
C04334=1109.265,388.460,409.314,-178.524,14.980,150.817
C04335=1109.271,388.706,409.278,-178.521,14.985,150.818
C04336=1109.276,388.953,409.240,-178.519,14.989,150.818
C04337=1109.282,389.201,409.203,-178.516,14.994,150.819
C04338=1109.288,389.448,409.166,-178.514,14.998,150.820
C04339=1109.293,389.694,409.130,-178.511,15.003,150.820
C04340=1109.299,389.942,409.093,-178.509,15.007,150.821
C04341=1109.304,390.189,409.056,-178.507,15.011,150.821
C04342=1109.310,390.436,409.019,-178.504,15.015,150.822
C04343=1109.316,390.683,408.983,-178.501,15.020,150.822
C04344=1109.322,390.929,408.945,-178.499,15.025,150.823
C04345=1109.327,391.177,408.908,-178.497,15.029,150.824
C04346=1109.333,391.424,408.871,-178.495,15.033,150.824
C04347=1109.338,391.672,408.834,-178.492,15.038,150.825
C04348=1109.345,391.919,408.798,-178.490,15.042,150.825
C04349=1109.350,392.166,408.761,-178.487,15.047,150.826
C04350=1109.356,392.413,408.724,-178.485,15.051,150.827
C04351=1109.362,392.660,408.686,-178.483,15.056,150.827
C04352=1109.367,392.907,408.649,-178.481,15.060,150.828
C04353=1109.373,393.154,408.612,-178.478,15.065,150.829
C04354=1109.378,393.402,408.575,-178.476,15.070,150.829
C04355=1109.384,393.649,408.538,-178.473,15.074,150.830
C04356=1109.390,393.896,408.500,-178.471,15.079,150.831
C04357=1109.395,394.143,408.463,-178.469,15.083,150.831
C04358=1109.401,394.390,408.426,-178.467,15.088,150.832
C04359=1109.407,394.637,408.389,-178.464,15.093,150.833
C04360=1109.412,394.884,408.352,-178.462,15.098,150.833
C04361=1109.417,395.131,408.315,-178.460,15.103,150.834
C04362=1109.423,395.378,408.278,-178.458,15.107,150.835
C04363=1109.429,395.625,408.240,-178.455,15.112,150.835
C04364=1109.434,395.873,408.203,-178.453,15.117,150.836
C04365=1109.440,396.119,408.165,-178.451,15.122,150.837
C04366=1109.445,396.331,408.134,-178.449,15.126,150.838
C04367=1109.451,396.543,408.102,-178.447,15.130,150.838
C04368=1109.455,396.755,408.070,-178.445,15.134,150.839
C04369=1109.460,396.966,408.038,-178.443,15.139,150.840
C04370=1109.464,397.179,408.005,-178.441,15.143,150.840
C04371=1109.469,397.390,407.973,-178.440,15.147,150.841
C04372=1109.475,397.602,407.942,-178.438,15.151,150.841
C04373=1109.479,397.814,407.909,-178.436,15.155,150.842
C04374=1109.484,398.061,407.872,-178.434,15.160,150.843
C04375=1109.490,398.308,407.834,-178.431,15.165,150.844
C04376=1109.496,398.555,407.797,-178.429,15.170,150.844
C04377=1109.502,398.802,407.759,-178.427,15.175,150.845
C04378=1109.507,399.050,407.722,-178.425,15.180,150.846
C04379=1109.513,399.296,407.684,-178.423,15.185,150.847
C04380=1109.518,399.543,407.646,-178.420,15.190,150.848
C04381=1109.524,399.790,407.609,-178.418,15.196,150.849
C04382=1109.530,400.037,407.571,-178.416,15.201,150.849
C04383=1109.535,400.285,407.534,-178.414,15.206,150.850
C04384=1109.541,400.532,407.496,-178.412,15.210,150.851
C04385=1109.547,400.778,407.458,-178.410,15.216,150.852
C04386=1109.552,401.026,407.421,-178.408,15.221,150.853
C04387=1109.557,401.273,407.383,-178.406,15.226,150.854
C04388=1109.563,401.520,407.345,-178.404,15.231,150.855
C04389=1109.568,401.767,407.308,-178.402,15.237,150.855
C04390=1109.574,402.014,407.270,-178.400,15.242,150.856
C04391=1109.580,402.261,407.232,-178.398,15.247,150.857
C04392=1109.585,402.508,407.194,-178.396,15.252,150.858
C04393=1109.591,402.755,407.157,-178.393,15.258,150.859
C04394=1109.597,403.003,407.119,-178.391,15.264,150.860
C04395=1109.602,403.250,407.080,-178.389,15.269,150.861
C04396=1109.608,403.496,407.042,-178.387,15.274,150.862
C04397=1109.614,403.744,407.005,-178.385,15.280,150.863
C04398=1109.619,403.991,406.967,-178.383,15.285,150.864
C04399=1109.625,404.238,406.929,-178.381,15.290,150.865
C04400=1109.630,404.485,406.891,-178.379,15.296,150.865
C04401=1109.636,404.731,406.853,-178.377,15.301,150.866
C04402=1109.643,404.979,406.815,-178.375,15.306,150.867
C04403=1109.648,405.226,406.777,-178.374,15.312,150.868
C04404=1109.654,405.473,406.739,-178.372,15.318,150.869
C04405=1109.659,405.720,406.701,-178.369,15.324,150.870
C04406=1109.664,405.967,406.664,-178.367,15.329,150.871
C04407=1109.670,406.214,406.625,-178.365,15.335,150.872
C04408=1109.675,406.461,406.587,-178.363,15.340,150.873
C04409=1109.681,406.708,406.549,-178.361,15.346,150.874
C04410=1109.687,406.955,406.511,-178.360,15.351,150.875
C04411=1109.692,407.202,406.473,-178.358,15.357,150.876
C04412=1109.698,407.449,406.434,-178.355,15.363,150.877
C04413=1109.704,407.696,406.396,-178.354,15.369,150.878
C04414=1109.709,407.943,406.357,-178.352,15.375,150.880
C04415=1109.715,408.189,406.320,-178.350,15.380,150.881
C04416=1109.721,408.437,406.281,-178.348,15.387,150.882
C04417=1109.726,408.684,406.243,-178.346,15.392,150.883
C04418=1109.732,408.931,406.205,-178.344,15.398,150.884
C04419=1109.737,409.178,406.167,-178.343,15.404,150.885
C04420=1109.742,409.425,406.128,-178.340,15.410,150.886
C04421=1109.749,409.672,406.089,-178.339,15.416,150.887
C04422=1109.753,409.883,406.057,-178.337,15.420,150.888
C04423=1109.757,410.095,406.024,-178.336,15.426,150.889
C04424=1109.762,410.307,405.991,-178.334,15.431,150.890
C04425=1109.767,410.518,405.958,-178.332,15.436,150.891
C04426=1109.772,410.729,405.925,-178.331,15.442,150.892
C04427=1109.777,410.941,405.893,-178.329,15.446,150.893
C04428=1109.782,411.152,405.859,-178.328,15.452,150.894
C04429=1109.786,411.364,405.826,-178.326,15.457,150.895
C04430=1109.791,411.611,405.788,-178.324,15.464,150.896
C04431=1109.798,411.858,405.749,-178.323,15.469,150.897
C04432=1109.803,412.105,405.711,-178.321,15.475,150.899
C04433=1109.808,412.352,405.672,-178.319,15.482,150.900
C04434=1109.814,412.598,405.633,-178.317,15.488,150.901
C04435=1109.820,412.846,405.595,-178.316,15.493,150.902
C04436=1109.826,413.093,405.557,-178.314,15.500,150.903
C04437=1109.831,413.339,405.518,-178.312,15.506,150.905
C04438=1109.836,413.586,405.480,-178.310,15.513,150.906
C04439=1109.842,413.833,405.440,-178.309,15.519,150.907
C04440=1109.847,414.080,405.402,-178.307,15.525,150.908
C04441=1109.854,414.326,405.363,-178.305,15.532,150.909
C04442=1109.859,414.574,405.325,-178.303,15.538,150.911
C04443=1109.865,414.821,405.285,-178.301,15.544,150.912
C04444=1109.870,415.068,405.247,-178.300,15.551,150.913
C04445=1109.876,415.315,405.208,-178.298,15.558,150.915
C04446=1109.881,415.562,405.169,-178.297,15.564,150.916
C04447=1109.888,415.808,405.131,-178.295,15.570,150.917
C04448=1109.893,416.056,405.092,-178.293,15.576,150.918
C04449=1109.899,416.302,405.053,-178.291,15.583,150.920
C04450=1109.904,416.549,405.014,-178.290,15.590,150.921
C04451=1109.910,416.796,404.975,-178.288,15.596,150.922
C04452=1109.915,417.043,404.936,-178.287,15.603,150.924
C04453=1109.921,417.289,404.897,-178.285,15.610,150.925
C04454=1109.927,417.537,404.858,-178.283,15.616,150.926
C04455=1109.932,417.783,404.819,-178.282,15.623,150.928
C04456=1109.938,418.030,404.780,-178.281,15.629,150.929
C04457=1109.943,418.278,404.742,-178.279,15.637,150.931
C04458=1109.949,418.524,404.703,-178.277,15.643,150.932
C04459=1109.955,418.771,404.663,-178.275,15.650,150.933
C04460=1109.960,419.018,404.624,-178.274,15.657,150.935
C04461=1109.966,419.265,404.586,-178.273,15.663,150.936
C04462=1109.971,419.512,404.546,-178.271,15.670,150.938
C04463=1109.976,419.759,404.507,-178.269,15.678,150.939
C04464=1109.982,420.005,404.468,-178.268,15.684,150.941
C04465=1109.988,420.252,404.428,-178.266,15.691,150.942
C04466=1109.993,420.499,404.389,-178.264,15.698,150.943
C04467=1109.999,420.746,404.350,-178.264,15.705,150.945
C04468=1110.005,420.993,404.311,-178.262,15.712,150.946
C04469=1110.010,421.239,404.272,-178.260,15.719,150.948
C04470=1110.016,421.486,404.233,-178.259,15.726,150.949
C04471=1110.021,421.733,404.193,-178.257,15.733,150.951
C04472=1110.027,421.980,404.154,-178.256,15.741,150.952
C04473=1110.033,422.227,404.115,-178.255,15.748,150.954
C04474=1110.039,422.474,404.075,-178.253,15.755,150.955
C04475=1110.044,422.720,404.036,-178.251,15.762,150.957
C04476=1110.050,422.967,403.997,-178.250,15.770,150.959
C04477=1110.055,423.214,403.957,-178.249,15.776,150.960
C04478=1110.061,423.432,403.922,-178.247,15.783,150.961
C04479=1110.065,423.649,403.888,-178.246,15.790,150.963
C04480=1110.070,423.867,403.853,-178.245,15.796,150.964
C04481=1110.075,424.085,403.818,-178.244,15.803,150.966
C04482=1110.080,424.303,403.783,-178.243,15.809,150.967
C04483=1110.084,424.520,403.748,-178.242,15.815,150.968
C04484=1110.089,424.739,403.713,-178.240,15.822,150.970
C04485=1110.094,424.957,403.678,-178.240,15.829,150.971
C04486=1110.100,425.204,403.639,-178.238,15.836,150.973
C04487=1110.105,425.450,403.598,-178.237,15.844,150.975
C04488=1110.111,425.696,403.559,-178.235,15.851,150.976
C04489=1110.117,425.943,403.520,-178.234,15.859,150.978
C04490=1110.121,426.190,403.480,-178.232,15.867,150.980
C04491=1110.128,426.437,403.441,-178.232,15.874,150.981
C04492=1110.133,426.683,403.401,-178.231,15.882,150.983
C04493=1110.139,426.931,403.361,-178.229,15.889,150.985
C04494=1110.144,427.177,403.322,-178.228,15.897,150.987
C04495=1110.150,427.424,403.281,-178.227,15.905,150.988
C04496=1110.155,427.670,403.242,-178.226,15.913,150.990
C04497=1110.161,427.917,403.203,-178.224,15.921,150.992
C04498=1110.166,428.164,403.162,-178.223,15.929,150.994
C04499=1110.172,428.411,403.123,-178.222,15.936,150.995
C04500=1110.178,428.658,403.082,-178.220,15.944,150.997
C04501=1110.184,428.904,403.043,-178.219,15.952,150.999
C04502=1110.189,429.151,403.002,-178.218,15.960,151.001
C04503=1110.195,429.397,402.963,-178.217,15.968,151.002
C04504=1110.200,429.645,402.923,-178.216,15.976,151.004
C04505=1110.206,429.890,402.884,-178.215,15.984,151.006
C04506=1110.211,430.138,402.844,-178.214,15.992,151.008
C04507=1110.217,430.384,402.804,-178.213,16.000,151.010
C04508=1110.223,430.631,402.763,-178.212,16.009,151.012
C04509=1110.228,430.877,402.724,-178.211,16.017,151.014
C04510=1110.234,431.124,402.683,-178.210,16.025,151.016
C04511=1110.238,431.371,402.644,-178.209,16.033,151.017
C04512=1110.245,431.617,402.603,-178.208,16.041,151.019
C04513=1110.250,431.865,402.563,-178.207,16.049,151.021
C04514=1110.256,432.110,402.524,-178.206,16.058,151.023
C04515=1110.262,432.357,402.483,-178.205,16.066,151.025
C04516=1110.266,432.604,402.443,-178.204,16.074,151.027
C04517=1110.273,432.850,402.403,-178.203,16.083,151.029
C04518=1110.278,433.097,402.363,-178.202,16.091,151.031
C04519=1110.283,433.343,402.322,-178.202,16.100,151.033
C04520=1110.289,433.590,402.282,-178.201,16.108,151.035
C04521=1110.294,433.837,402.242,-178.199,16.117,151.037
C04522=1110.300,434.083,402.201,-178.198,16.126,151.039
C04523=1110.306,434.329,402.162,-178.198,16.134,151.041
C04524=1110.311,434.577,402.122,-178.197,16.143,151.043
C04525=1110.317,434.824,402.081,-178.196,16.151,151.045
C04526=1110.322,435.070,402.040,-178.196,16.160,151.047
C04527=1110.328,435.316,402.000,-178.194,16.169,151.049
C04528=1110.333,435.562,401.960,-178.194,16.178,151.052
C04529=1110.339,435.809,401.919,-178.193,16.187,151.054
C04530=1110.345,436.056,401.878,-178.193,16.195,151.056
C04531=1110.349,436.303,401.839,-178.192,16.204,151.058
C04532=1110.355,436.549,401.798,-178.191,16.213,151.060
C04533=1110.360,436.796,401.758,-178.190,16.222,151.062
C04534=1110.366,437.028,401.720,-178.189,16.231,151.064
C04535=1110.371,437.261,401.681,-178.189,16.239,151.066
C04536=1110.377,437.492,401.643,-178.189,16.247,151.068
C04537=1110.382,437.725,401.604,-178.188,16.256,151.070
C04538=1110.387,437.958,401.566,-178.187,16.265,151.073
C04539=1110.392,438.190,401.528,-178.187,16.273,151.075
C04540=1110.397,438.423,401.489,-178.186,16.282,151.077
C04541=1110.403,438.656,401.451,-178.186,16.290,151.079
C04542=1110.408,438.902,401.411,-178.185,16.299,151.081
C04543=1110.413,439.149,401.370,-178.184,16.309,151.083
C04544=1110.419,439.396,401.329,-178.184,16.318,151.086
C04545=1110.425,439.642,401.289,-178.184,16.327,151.088
C04546=1110.430,439.889,401.248,-178.183,16.337,151.090
C04547=1110.436,440.135,401.207,-178.182,16.346,151.093
C04548=1110.441,440.382,401.166,-178.182,16.356,151.095
C04549=1110.447,440.628,401.125,-178.181,16.365,151.097
C04550=1110.452,440.875,401.085,-178.181,16.375,151.100
C04551=1110.458,441.121,401.044,-178.181,16.384,151.102
C04552=1110.464,441.368,401.003,-178.180,16.394,151.104
C04553=1110.469,441.614,400.962,-178.180,16.403,151.107
C04554=1110.474,441.861,400.922,-178.179,16.413,151.109
C04555=1110.480,442.107,400.880,-178.179,16.423,151.112
C04556=1110.485,442.353,400.840,-178.179,16.432,151.114
C04557=1110.491,442.600,400.799,-178.178,16.443,151.117
C04558=1110.497,442.846,400.758,-178.178,16.452,151.119
C04559=1110.503,443.093,400.717,-178.178,16.462,151.122
C04560=1110.508,443.338,400.676,-178.178,16.472,151.124
C04561=1110.513,443.585,400.635,-178.178,16.482,151.127
C04562=1110.518,443.832,400.594,-178.177,16.492,151.129
C04563=1110.524,444.078,400.553,-178.177,16.502,151.132
C04564=1110.529,444.325,400.512,-178.177,16.512,151.134
C04565=1110.535,444.571,400.470,-178.178,16.522,151.137
C04566=1110.540,444.818,400.429,-178.178,16.532,151.140
C04567=1110.546,445.064,400.388,-178.179,16.540,151.142
C04568=1110.551,445.310,400.347,-178.180,16.551,151.145
C04569=1110.557,445.556,400.306,-178.180,16.561,151.148
C04570=1110.563,445.803,400.265,-178.181,16.570,151.150
C04571=1110.568,446.050,400.223,-178.182,16.580,151.153
C04572=1110.574,446.297,400.182,-178.183,16.590,151.156
C04573=1110.580,446.543,400.141,-178.184,16.599,151.158
C04574=1110.584,446.789,400.100,-178.186,16.609,151.161
C04575=1110.590,447.035,400.058,-178.187,16.619,151.164
C04576=1110.596,447.282,400.018,-178.188,16.628,151.167
C04577=1110.601,447.529,399.976,-178.190,16.638,151.170
C04578=1110.606,447.776,399.935,-178.191,16.648,151.172
C04579=1110.612,448.021,399.894,-178.193,16.658,151.175
C04580=1110.617,448.268,399.852,-178.195,16.667,151.178
C04581=1110.623,448.514,399.811,-178.196,16.677,151.181
C04582=1110.628,448.761,399.769,-178.198,16.686,151.184
C04583=1110.633,449.008,399.728,-178.200,16.696,151.187
C04584=1110.639,449.254,399.687,-178.202,16.705,151.190
C04585=1110.645,449.500,399.645,-178.205,16.714,151.192
C04586=1110.650,449.747,399.604,-178.206,16.725,151.195
C04587=1110.656,449.993,399.563,-178.209,16.734,151.198
C04588=1110.661,450.239,399.521,-178.211,16.743,151.201
C04589=1110.666,450.486,399.480,-178.214,16.753,151.204
C04590=1110.255,450.480,399.378,-178.302,16.987,151.283
C04591=1110.250,450.233,399.419,-178.299,16.977,151.280
C04592=1110.245,449.988,399.460,-178.297,16.968,151.277
C04593=1110.239,449.742,399.502,-178.295,16.958,151.274
C04594=1110.234,449.495,399.544,-178.293,16.948,151.271
C04595=1110.228,449.248,399.585,-178.291,16.939,151.268
C04596=1110.223,449.002,399.627,-178.289,16.929,151.265
C04597=1110.217,448.756,399.668,-178.287,16.919,151.262
C04598=1110.211,448.509,399.709,-178.285,16.910,151.259
C04599=1110.206,448.262,399.751,-178.283,16.900,151.256
C04600=1110.200,448.016,399.792,-178.282,16.890,151.253
C04601=1110.196,447.770,399.833,-178.280,16.881,151.251
C04602=1110.190,447.523,399.875,-178.278,16.871,151.248
C04603=1110.184,447.277,399.916,-178.277,16.861,151.245
C04604=1110.179,447.030,399.958,-178.275,16.851,151.242
C04605=1110.173,446.784,399.999,-178.274,16.841,151.239
C04606=1110.168,446.537,400.040,-178.273,16.832,151.237
C04607=1110.163,446.291,400.082,-178.272,16.821,151.234
C04608=1110.157,446.045,400.123,-178.271,16.812,151.231
C04609=1110.151,445.798,400.164,-178.270,16.802,151.228
C04610=1110.146,445.552,400.206,-178.269,16.792,151.226
C04611=1110.140,445.305,400.247,-178.268,16.782,151.223
C04612=1110.134,445.059,400.288,-178.268,16.773,151.220
C04613=1110.129,444.813,400.328,-178.268,16.763,151.218
C04614=1110.124,444.566,400.370,-178.267,16.753,151.215
C04615=1110.119,444.319,400.411,-178.267,16.743,151.212
C04616=1110.113,444.073,400.453,-178.267,16.733,151.210
C04617=1110.107,443.826,400.493,-178.267,16.723,151.207
C04618=1110.102,443.580,400.535,-178.267,16.713,151.205
C04619=1110.097,443.334,400.576,-178.266,16.703,151.202
C04620=1110.091,443.087,400.617,-178.267,16.693,151.200
C04621=1110.085,442.841,400.658,-178.267,16.683,151.197
C04622=1110.080,442.595,400.699,-178.268,16.673,151.195
C04623=1110.074,442.348,400.740,-178.268,16.663,151.192
C04624=1110.068,442.101,400.781,-178.269,16.653,151.190
C04625=1110.063,441.855,400.822,-178.269,16.644,151.187
C04626=1110.058,441.609,400.863,-178.270,16.633,151.185
C04627=1110.053,441.362,400.904,-178.270,16.624,151.182
C04628=1110.047,441.116,400.945,-178.270,16.615,151.180
C04629=1110.041,440.869,400.986,-178.271,16.604,151.177
C04630=1110.036,440.623,401.026,-178.271,16.595,151.175
C04631=1110.030,440.377,401.068,-178.272,16.585,151.173
C04632=1110.024,440.130,401.109,-178.272,16.576,151.170
C04633=1110.019,439.884,401.149,-178.272,16.567,151.168
C04634=1110.014,439.637,401.190,-178.273,16.557,151.166
C04635=1110.008,439.390,401.230,-178.274,16.547,151.163
C04636=1110.002,439.144,401.272,-178.274,16.539,151.161
C04637=1109.996,438.898,401.312,-178.275,16.529,151.159
C04638=1109.991,438.651,401.352,-178.276,16.519,151.157
C04639=1109.985,438.420,401.391,-178.276,16.511,151.155
C04640=1109.980,438.188,401.429,-178.277,16.502,151.152
C04641=1109.975,437.956,401.467,-178.278,16.493,151.150
C04642=1109.970,437.724,401.505,-178.278,16.485,151.148
C04643=1109.965,437.493,401.543,-178.279,16.476,151.146
C04644=1109.959,437.261,401.581,-178.280,16.467,151.144
C04645=1109.954,437.030,401.620,-178.280,16.459,151.142
C04646=1109.949,436.798,401.657,-178.281,16.451,151.140
C04647=1109.943,436.551,401.698,-178.282,16.441,151.138
C04648=1109.938,436.304,401.739,-178.282,16.432,151.136
C04649=1109.933,436.058,401.779,-178.283,16.423,151.133
C04650=1109.927,435.811,401.820,-178.284,16.415,151.131
C04651=1109.922,435.565,401.860,-178.285,16.405,151.129
C04652=1109.916,435.318,401.901,-178.285,16.396,151.127
C04653=1109.910,435.072,401.941,-178.286,16.388,151.125
C04654=1109.905,434.825,401.982,-178.287,16.379,151.123
C04655=1109.899,434.579,402.022,-178.288,16.371,151.121
C04656=1109.894,434.333,402.063,-178.289,16.361,151.119
C04657=1109.888,434.085,402.102,-178.290,16.353,151.117
C04658=1109.883,433.839,402.143,-178.291,16.344,151.115
C04659=1109.878,433.592,402.183,-178.291,16.335,151.112
C04660=1109.872,433.346,402.224,-178.292,16.327,151.111
C04661=1109.866,433.100,402.264,-178.293,16.319,151.109
C04662=1109.861,432.852,402.304,-178.295,16.309,151.106
C04663=1109.855,432.606,402.345,-178.295,16.301,151.104
C04664=1109.849,432.360,402.384,-178.296,16.293,151.103
C04665=1109.844,432.112,402.424,-178.297,16.284,151.101
C04666=1109.839,431.866,402.465,-178.298,16.276,151.099
C04667=1109.833,431.620,402.505,-178.299,16.268,151.097
C04668=1109.827,431.372,402.545,-178.300,16.259,151.095
C04669=1109.822,431.126,402.585,-178.301,16.251,151.093
C04670=1109.816,430.880,402.626,-178.302,16.243,151.091
C04671=1109.811,430.633,402.665,-178.303,16.234,151.089
C04672=1109.805,430.386,402.705,-178.304,16.226,151.087
C04673=1109.800,430.140,402.746,-178.305,16.218,151.085
C04674=1109.794,429.893,402.785,-178.306,16.210,151.083
C04675=1109.789,429.647,402.826,-178.308,16.202,151.082
C04676=1109.783,429.399,402.866,-178.309,16.194,151.080
C04677=1109.777,429.153,402.906,-178.310,16.186,151.078
C04678=1109.771,428.907,402.945,-178.311,16.178,151.076
C04679=1109.766,428.660,402.986,-178.312,16.170,151.074
C04680=1109.760,428.413,403.025,-178.313,16.162,151.073
C04681=1109.755,428.166,403.065,-178.315,16.154,151.071
C04682=1109.749,427.920,403.104,-178.316,16.146,151.069
C04683=1109.744,427.673,403.144,-178.317,16.138,151.067
C04684=1109.738,427.427,403.184,-178.318,16.130,151.065
C04685=1109.732,427.180,403.224,-178.320,16.122,151.064
C04686=1109.727,426.932,403.264,-178.321,16.114,151.062
C04687=1109.721,426.686,403.303,-178.322,16.107,151.060
C04688=1109.716,426.439,403.343,-178.324,16.099,151.058
C04689=1109.710,426.192,403.383,-178.325,16.091,151.057
C04690=1109.704,425.946,403.423,-178.326,16.083,151.055
C04691=1109.699,425.699,403.462,-178.328,16.076,151.053
C04692=1109.693,425.452,403.502,-178.328,16.069,151.052
C04693=1109.688,425.205,403.541,-178.330,16.061,151.050
C04694=1109.682,424.960,403.581,-178.331,16.053,151.048
C04695=1109.678,424.741,403.616,-178.332,16.047,151.047
C04696=1109.673,424.523,403.651,-178.334,16.040,151.046
C04697=1109.668,424.305,403.686,-178.335,16.033,151.044
C04698=1109.663,424.087,403.721,-178.336,16.026,151.043
C04699=1109.658,423.869,403.756,-178.338,16.020,151.041
C04700=1109.653,423.651,403.791,-178.338,16.013,151.040
C04701=1109.648,423.433,403.826,-178.340,16.007,151.038
C04702=1109.644,423.215,403.860,-178.341,16.000,151.037
C04703=1109.637,422.969,403.900,-178.342,15.993,151.035
C04704=1109.632,422.722,403.939,-178.344,15.985,151.034
C04705=1109.626,422.475,403.979,-178.346,15.978,151.032
C04706=1109.620,422.229,404.018,-178.347,15.971,151.031
C04707=1109.615,421.981,404.058,-178.348,15.964,151.029
C04708=1109.609,421.735,404.097,-178.350,15.956,151.028
C04709=1109.603,421.488,404.136,-178.352,15.949,151.026
C04710=1109.598,421.241,404.175,-178.353,15.942,151.025
C04711=1109.592,420.995,404.215,-178.354,15.935,151.023
C04712=1109.586,420.748,404.254,-178.356,15.928,151.022
C04713=1109.582,420.501,404.294,-178.357,15.921,151.020
C04714=1109.576,420.253,404.332,-178.359,15.914,151.019
C04715=1109.570,420.007,404.371,-178.360,15.907,151.017
C04716=1109.564,419.760,404.411,-178.362,15.900,151.016
C04717=1109.559,419.513,404.450,-178.364,15.893,151.014
C04718=1109.553,419.267,404.489,-178.365,15.886,151.013
C04719=1109.547,419.020,404.528,-178.366,15.879,151.011
C04720=1109.542,418.773,404.567,-178.368,15.872,151.010
C04721=1109.537,418.526,404.606,-178.370,15.865,151.008
C04722=1109.531,418.279,404.645,-178.371,15.859,151.007
C04723=1109.525,418.033,404.684,-178.373,15.852,151.006
C04724=1109.520,417.785,404.724,-178.375,15.844,151.004
C04725=1109.515,417.538,404.763,-178.376,15.838,151.003
C04726=1109.509,417.292,404.802,-178.378,15.831,151.001
C04727=1109.503,417.045,404.841,-178.379,15.825,151.000
C04728=1109.498,416.797,404.880,-178.381,15.817,150.999
C04729=1109.492,416.551,404.919,-178.383,15.811,150.997
C04730=1109.486,416.304,404.957,-178.384,15.804,150.996
C04731=1109.480,416.057,404.996,-178.387,15.798,150.995
C04732=1109.475,415.811,405.035,-178.388,15.791,150.993
C04733=1109.469,415.564,405.074,-178.390,15.784,150.992
C04734=1109.464,415.317,405.113,-178.391,15.778,150.991
C04735=1109.458,415.070,405.152,-178.393,15.771,150.989
C04736=1109.452,414.822,405.190,-178.395,15.765,150.988
C04737=1109.447,414.576,405.229,-178.397,15.758,150.987
C04738=1109.441,414.329,405.267,-178.398,15.752,150.986
C04739=1109.435,414.082,405.307,-178.400,15.746,150.985
C04740=1109.430,413.835,405.345,-178.402,15.739,150.983
C04741=1109.424,413.589,405.384,-178.403,15.733,150.982
C04742=1109.419,413.341,405.423,-178.405,15.727,150.981
C04743=1109.413,413.094,405.462,-178.407,15.720,150.979
C04744=1109.407,412.848,405.500,-178.409,15.714,150.978
C04745=1109.401,412.600,405.539,-178.411,15.708,150.977
C04746=1109.396,412.353,405.577,-178.412,15.702,150.976
C04747=1109.391,412.106,405.616,-178.414,15.695,150.975
C04748=1109.385,411.860,405.654,-178.416,15.689,150.973
C04749=1109.379,411.612,405.693,-178.418,15.683,150.972
C04750=1109.374,411.365,405.731,-178.420,15.677,150.971
C04751=1109.369,411.155,405.765,-178.421,15.671,150.970
C04752=1109.364,410.943,405.798,-178.423,15.666,150.969
C04753=1109.359,410.730,405.831,-178.425,15.661,150.968
C04754=1109.355,410.520,405.864,-178.426,15.656,150.967
C04755=1109.349,410.308,405.896,-178.428,15.650,150.966
C04756=1109.345,410.096,405.929,-178.429,15.646,150.965
C04757=1109.340,409.884,405.962,-178.431,15.640,150.964
C04758=1109.335,409.673,405.995,-178.433,15.635,150.963
C04759=1109.330,409.426,406.034,-178.434,15.629,150.962
C04760=1109.324,409.179,406.072,-178.436,15.623,150.961
C04761=1109.319,408.932,406.110,-178.438,15.617,150.960
C04762=1109.313,408.685,406.149,-178.440,15.611,150.959
C04763=1109.307,408.438,406.186,-178.442,15.605,150.957
C04764=1109.302,408.192,406.225,-178.443,15.599,150.956
C04765=1109.297,407.945,406.264,-178.446,15.593,150.955
C04766=1109.290,407.697,406.302,-178.448,15.587,150.954
C04767=1109.285,407.450,406.340,-178.449,15.582,150.953
C04768=1109.279,407.203,406.378,-178.451,15.576,150.952
C04769=1109.274,406.956,406.416,-178.453,15.571,150.951
C04770=1109.269,406.709,406.455,-178.455,15.564,150.950
C04771=1109.263,406.463,406.492,-178.457,15.558,150.949
C04772=1109.257,406.215,406.531,-178.459,15.553,150.948
C04773=1109.251,405.968,406.569,-178.461,15.547,150.947
C04774=1109.246,405.721,406.607,-178.463,15.542,150.946
C04775=1109.240,405.474,406.645,-178.466,15.536,150.945
C04776=1109.235,405.227,406.683,-178.467,15.530,150.944
C04777=1109.229,404.980,406.721,-178.469,15.525,150.943
C04778=1109.223,404.733,406.760,-178.471,15.519,150.942
C04779=1109.218,404.486,406.798,-178.473,15.514,150.941
C04780=1109.212,404.239,406.835,-178.475,15.508,150.940
C04781=1109.207,403.992,406.873,-178.477,15.503,150.939
C04782=1109.201,403.745,406.911,-178.479,15.497,150.938
C04783=1109.196,403.498,406.949,-178.482,15.491,150.937
C04784=1109.190,403.251,406.987,-178.484,15.486,150.936
C04785=1109.184,403.004,407.025,-178.486,15.481,150.935
C04786=1109.178,402.756,407.063,-178.487,15.475,150.934
C04787=1109.173,402.509,407.100,-178.489,15.470,150.933
C04788=1109.167,402.262,407.138,-178.491,15.464,150.933
C04789=1109.161,402.015,407.176,-178.494,15.459,150.932
C04790=1109.156,401.769,407.214,-178.496,15.454,150.931
C04791=1109.151,401.521,407.252,-178.498,15.449,150.930
C04792=1109.145,401.274,407.290,-178.500,15.443,150.929
C04793=1109.139,401.027,407.327,-178.502,15.438,150.928
C04794=1109.133,400.780,407.364,-178.504,15.433,150.927
C04795=1109.128,400.533,407.403,-178.506,15.427,150.926
C04796=1109.122,400.286,407.440,-178.508,15.422,150.926
C04797=1109.117,400.039,407.477,-178.510,15.417,150.925
C04798=1109.111,399.792,407.516,-178.512,15.412,150.924
C04799=1109.106,399.545,407.554,-178.515,15.407,150.923
C04800=1109.100,399.298,407.591,-178.517,15.401,150.922
C04801=1109.094,399.051,407.628,-178.519,15.397,150.921
C04802=1109.088,398.804,407.665,-178.521,15.391,150.920
C04803=1109.083,398.557,407.704,-178.524,15.386,150.920
C04804=1109.078,398.309,407.741,-178.526,15.381,150.919
C04805=1109.072,398.062,407.779,-178.528,15.376,150.918
C04806=1109.066,397.815,407.816,-178.530,15.371,150.917
C04807=1109.061,397.603,407.849,-178.532,15.367,150.917
C04808=1109.056,397.392,407.881,-178.533,15.362,150.916
C04809=1109.051,397.179,407.912,-178.535,15.359,150.915
C04810=1109.047,396.968,407.945,-178.537,15.354,150.915
C04811=1109.042,396.756,407.976,-178.540,15.350,150.914
C04812=1109.037,396.544,408.009,-178.541,15.345,150.913
C04813=1109.032,396.332,408.041,-178.543,15.342,150.913
C04814=1109.027,396.121,408.073,-178.545,15.337,150.912
C04815=1109.021,395.873,408.110,-178.547,15.332,150.911
C04816=1109.017,395.626,408.147,-178.550,15.327,150.910
C04817=1109.011,395.380,408.185,-178.552,15.322,150.910
C04818=1109.005,395.132,408.222,-178.554,15.317,150.909
C04819=1109.000,394.885,408.259,-178.556,15.313,150.908
C04820=1108.994,394.638,408.297,-178.558,15.309,150.908
C04821=1108.988,394.391,408.334,-178.561,15.304,150.907
C04822=1108.983,394.143,408.371,-178.563,15.299,150.906
C04823=1108.977,393.897,408.409,-178.565,15.294,150.905
C04824=1108.971,393.649,408.446,-178.568,15.289,150.905
C04825=1108.966,393.402,408.483,-178.570,15.285,150.904
C04826=1108.959,393.155,408.519,-178.572,15.280,150.903
C04827=1108.954,392.909,408.557,-178.575,15.275,150.903
C04828=1108.948,392.661,408.594,-178.577,15.270,150.902
C04829=1108.943,392.414,408.631,-178.580,15.266,150.901
C04830=1108.937,392.167,408.668,-178.581,15.261,150.901
C04831=1108.932,391.919,408.705,-178.584,15.257,150.900
C04832=1108.926,391.673,408.743,-178.587,15.252,150.900
C04833=1108.920,391.425,408.780,-178.589,15.247,150.899
C04834=1108.914,391.178,408.816,-178.591,15.243,150.898
C04835=1108.909,390.931,408.853,-178.593,15.239,150.898
C04836=1108.903,390.684,408.890,-178.596,15.234,150.897
C04837=1108.898,390.437,408.927,-178.598,15.229,150.896
C04838=1108.892,390.189,408.964,-178.600,15.225,150.896
C04839=1108.886,389.942,409.000,-178.603,15.221,150.895
C04840=1108.880,389.696,409.038,-178.606,15.216,150.895
C04841=1108.875,389.449,409.075,-178.608,15.211,150.894
C04842=1108.869,389.202,409.112,-178.610,15.207,150.893
C04843=1108.863,388.955,409.148,-178.613,15.203,150.893
C04844=1108.857,388.707,409.185,-178.616,15.198,150.892
C04845=1108.852,388.460,409.222,-178.618,15.194,150.892
C04846=1108.846,388.213,409.258,-178.620,15.190,150.891
C04847=1108.840,387.966,409.295,-178.623,15.185,150.891
C04848=1108.835,387.718,409.332,-178.626,15.181,150.890
C04849=1108.830,387.471,409.368,-178.628,15.177,150.890
C04850=1108.824,387.224,409.405,-178.630,15.172,150.889
C04851=1108.818,386.977,409.442,-178.633,15.168,150.888
C04852=1108.812,386.730,409.479,-178.636,15.164,150.888
C04853=1108.807,386.483,409.515,-178.638,15.160,150.887
C04854=1108.801,386.236,409.552,-178.640,15.155,150.887
C04855=1108.796,385.989,409.589,-178.643,15.150,150.886
C04856=1108.789,385.741,409.625,-178.645,15.147,150.886
C04857=1108.784,385.494,409.661,-178.648,15.142,150.885
C04858=1108.779,385.247,409.698,-178.651,15.138,150.885
C04859=1108.773,385.000,409.735,-178.653,15.134,150.884
C04860=1108.768,384.753,409.772,-178.656,15.130,150.884
C04861=1108.762,384.505,409.807,-178.658,15.126,150.883
C04862=1108.757,384.259,409.844,-178.661,15.122,150.883
C04863=1108.747,383.847,409.905,-178.665,15.115,150.882
C04864=1108.738,383.435,409.966,-178.669,15.108,150.881
C04865=1108.729,383.023,410.027,-178.673,15.101,150.881
C04866=1108.719,382.612,410.087,-178.678,15.094,150.880
C04867=1108.713,382.364,410.123,-178.680,15.091,150.879
C04868=1108.708,382.117,410.160,-178.683,15.086,150.879
C04869=1108.702,381.870,410.196,-178.685,15.083,150.879
C04870=1108.696,381.623,410.232,-178.688,15.079,150.878
C04871=1108.691,381.376,410.268,-178.691,15.074,150.878
C04872=1108.685,381.128,410.304,-178.693,15.071,150.877
C04873=1108.679,380.881,410.341,-178.696,15.067,150.877
C04874=1108.674,380.634,410.377,-178.699,15.063,150.877
C04875=1108.667,380.387,410.413,-178.702,15.059,150.876
C04876=1108.663,380.140,410.449,-178.704,15.055,150.876
C04877=1108.656,379.893,410.485,-178.707,15.051,150.875
C04878=1108.650,379.645,410.521,-178.709,15.048,150.875
C04879=1108.645,379.398,410.558,-178.712,15.044,150.875
C04880=1108.639,379.151,410.594,-178.715,15.040,150.874
C04881=1108.634,378.903,410.631,-178.717,15.036,150.874
C04882=1108.628,378.656,410.666,-178.720,15.032,150.873
C04883=1108.622,378.409,410.702,-178.723,15.029,150.873
C04884=1108.617,378.162,410.738,-178.725,15.025,150.873
C04885=1108.611,377.914,410.774,-178.728,15.021,150.872
C04886=1108.606,377.667,410.810,-178.731,15.018,150.872
C04887=1108.600,377.420,410.847,-178.734,15.013,150.872
C04888=1108.594,377.172,410.882,-178.736,15.010,150.871
C04889=1108.589,376.925,410.918,-178.739,15.006,150.871
C04890=1108.583,376.678,410.953,-178.741,15.002,150.871
C04891=1108.578,376.431,410.990,-178.745,14.999,150.870
C04892=1108.571,376.183,411.026,-178.747,14.995,150.870
C04893=1108.566,375.936,411.061,-178.750,14.991,150.870
C04894=1108.561,375.688,411.097,-178.752,14.988,150.869
C04895=1108.555,375.442,411.134,-178.756,14.984,150.869
C04896=1108.549,375.194,411.169,-178.758,14.980,150.869
C04897=1108.544,374.947,411.205,-178.761,14.977,150.869
C04898=1108.538,374.699,411.241,-178.764,14.973,150.868
C04899=1108.533,374.452,411.276,-178.766,14.970,150.868
C04900=1108.527,374.205,411.312,-178.769,14.966,150.868
C04901=1108.521,373.958,411.347,-178.772,14.963,150.867
C04902=1108.515,373.711,411.384,-178.775,14.959,150.867
C04903=1108.510,373.464,411.419,-178.778,14.956,150.867
C04904=1108.504,373.216,411.455,-178.780,14.952,150.867
C04905=1108.498,372.969,411.490,-178.784,14.949,150.867
C04906=1108.492,372.721,411.526,-178.786,14.945,150.866
C04907=1108.487,372.474,411.561,-178.789,14.941,150.866
C04908=1108.481,372.226,411.598,-178.792,14.938,150.866
C04909=1108.476,371.979,411.633,-178.794,14.935,150.865
C04910=1108.470,371.732,411.669,-178.797,14.931,150.865
C04911=1108.465,371.485,411.704,-178.800,14.928,150.865
C04912=1108.458,371.237,411.740,-178.803,14.925,150.865
C04913=1108.453,370.990,411.775,-178.806,14.921,150.865
C04914=1108.447,370.742,411.811,-178.809,14.918,150.864
C04915=1108.439,370.357,411.866,-178.813,14.913,150.864
C04916=1108.430,369.972,411.921,-178.818,14.907,150.864
C04917=1108.420,369.587,411.976,-178.822,14.903,150.863
C04918=1108.412,369.202,412.031,-178.826,14.897,150.863
C04919=1108.407,368.955,412.066,-178.829,14.894,150.863
C04920=1108.400,368.707,412.101,-178.832,14.890,150.863
C04921=1108.395,368.460,412.137,-178.835,14.887,150.863
C04922=1108.389,368.212,412.173,-178.838,14.884,150.862
C04923=1108.384,367.966,412.208,-178.841,14.880,150.862
C04924=1108.378,367.718,412.243,-178.844,14.878,150.862
C04925=1108.372,367.470,412.278,-178.846,14.874,150.862
C04926=1108.367,367.223,412.314,-178.850,14.871,150.862
C04927=1108.361,366.975,412.349,-178.853,14.868,150.862
C04928=1108.356,366.728,412.384,-178.855,14.865,150.862
C04929=1108.350,366.481,412.419,-178.859,14.861,150.861
C04930=1108.345,366.233,412.454,-178.861,14.858,150.861
C04931=1108.339,365.986,412.489,-178.864,14.855,150.861
C04932=1108.333,365.739,412.525,-178.867,14.852,150.861
C04933=1108.327,365.491,412.560,-178.870,14.849,150.861
C04934=1108.322,365.244,412.595,-178.873,14.846,150.861
C04935=1108.316,364.996,412.630,-178.876,14.843,150.861
C04936=1108.310,364.749,412.665,-178.879,14.840,150.860
C04937=1108.305,364.501,412.699,-178.882,14.836,150.860
C04938=1108.299,364.254,412.735,-178.885,14.833,150.860
C04939=1108.294,364.006,412.770,-178.888,14.831,150.860
C04940=1108.288,363.759,412.804,-178.891,14.828,150.860
C04941=1108.282,363.511,412.840,-178.894,14.824,150.860
C04942=1108.276,363.264,412.875,-178.897,14.821,150.860
C04943=1108.271,363.016,412.910,-178.900,14.818,150.860
C04944=1108.265,362.769,412.945,-178.903,14.816,150.860
C04945=1108.259,362.522,412.979,-178.906,14.812,150.860
C04946=1108.254,362.275,413.015,-178.909,14.809,150.860
C04947=1108.248,362.027,413.049,-178.912,14.807,150.860
C04948=1108.242,361.779,413.084,-178.915,14.804,150.860
C04949=1108.237,361.532,413.119,-178.918,14.801,150.859
C04950=1108.231,361.284,413.154,-178.921,14.798,150.859
C04951=1108.225,361.036,413.188,-178.924,14.795,150.859
C04952=1108.220,360.789,413.224,-178.927,14.792,150.859
C04953=1108.214,360.542,413.258,-178.930,14.789,150.859
C04954=1108.208,360.294,413.293,-178.933,14.786,150.859
C04955=1108.202,360.047,413.327,-178.937,14.783,150.859
C04956=1108.197,359.800,413.362,-178.939,14.780,150.859
C04957=1108.191,359.551,413.397,-178.943,14.778,150.859
C04958=1108.186,359.304,413.431,-178.946,14.775,150.859
C04959=1108.180,359.057,413.466,-178.948,14.772,150.859
C04960=1108.174,358.810,413.500,-178.951,14.769,150.859
C04961=1108.169,358.561,413.536,-178.955,14.767,150.859
C04962=1108.163,358.314,413.570,-178.958,14.763,150.859
C04963=1108.158,358.067,413.604,-178.961,14.761,150.859
C04964=1108.152,357.819,413.638,-178.964,14.758,150.859
C04965=1108.146,357.572,413.674,-178.967,14.755,150.859
C04966=1108.140,357.324,413.708,-178.970,14.753,150.859
C04967=1108.132,356.954,413.760,-178.975,14.749,150.859
C04968=1108.123,356.584,413.811,-178.980,14.744,150.859
C04969=1108.115,356.214,413.862,-178.984,14.740,150.859
C04970=1108.107,355.843,413.914,-178.989,14.736,150.859
C04971=1108.101,355.595,413.948,-178.992,14.734,150.859
C04972=1108.095,355.348,413.982,-178.995,14.731,150.859
C04973=1108.089,355.100,414.017,-178.998,14.728,150.859
C04974=1108.083,354.853,414.051,-179.001,14.726,150.859
C04975=1108.078,354.605,414.086,-179.004,14.723,150.859
C04976=1108.072,354.358,414.120,-179.008,14.720,150.859
C04977=1108.067,354.110,414.155,-179.011,14.718,150.860
C04978=1108.061,353.863,414.189,-179.014,14.715,150.859
C04979=1108.055,353.615,414.223,-179.017,14.712,150.860
C04980=1108.050,353.367,414.258,-179.020,14.710,150.860
C04981=1108.044,353.119,414.291,-179.023,14.707,150.860
C04982=1108.038,352.872,414.325,-179.027,14.705,150.860
C04983=1108.033,352.624,414.360,-179.030,14.702,150.860
C04984=1108.027,352.377,414.394,-179.033,14.700,150.860
C04985=1108.021,352.129,414.428,-179.036,14.697,150.860
C04986=1108.015,351.882,414.462,-179.039,14.695,150.860
C04987=1108.010,351.634,414.496,-179.042,14.692,150.860
C04988=1108.004,351.386,414.530,-179.045,14.690,150.860
C04989=1107.999,351.139,414.564,-179.049,14.688,150.860
C04990=1107.993,350.892,414.599,-179.052,14.685,150.861
C04991=1107.988,350.644,414.632,-179.055,14.683,150.861
C04992=1107.982,350.396,414.667,-179.058,14.680,150.861
C04993=1107.976,350.148,414.701,-179.061,14.678,150.861
C04994=1107.970,349.900,414.734,-179.065,14.674,150.861
C04995=1107.965,349.653,414.769,-179.068,14.672,150.861
C04996=1107.959,349.406,414.803,-179.072,14.670,150.861
C04997=1107.953,349.158,414.836,-179.075,14.667,150.861
C04998=1107.948,348.910,414.870,-179.078,14.665,150.861
C04999=1107.942,348.663,414.904,-179.081,14.662,150.861
C05000=1107.936,348.415,414.938,-179.084,14.660,150.862
C05001=1107.931,348.168,414.972,-179.088,14.658,150.862
C05002=1107.926,347.920,415.006,-179.091,14.656,150.862
C05003=1107.920,347.672,415.040,-179.094,14.653,150.862
C05004=1107.914,347.425,415.073,-179.098,14.651,150.862
C05005=1107.908,347.177,415.107,-179.101,14.648,150.862
C05006=1107.903,346.929,415.141,-179.104,14.646,150.862
C05007=1107.897,346.682,415.175,-179.107,14.644,150.863
C05008=1107.891,346.433,415.208,-179.110,14.641,150.863
C05009=1107.885,346.186,415.242,-179.113,14.640,150.863
C05010=1107.880,345.938,415.276,-179.116,14.637,150.863
C05011=1107.874,345.691,415.310,-179.120,14.635,150.863
C05012=1107.869,345.443,415.344,-179.123,14.633,150.863
C05013=1107.863,345.195,415.378,-179.126,14.631,150.864
C05014=1107.857,344.948,415.411,-179.130,14.628,150.864
C05015=1107.852,344.700,415.444,-179.133,14.626,150.864
C05016=1107.846,344.452,415.478,-179.136,14.624,150.864
C05017=1107.840,344.204,415.512,-179.140,14.621,150.864
C05018=1107.835,343.957,415.545,-179.143,14.619,150.865
C05019=1107.826,343.589,415.595,-179.148,14.616,150.865
C05020=1107.818,343.221,415.645,-179.153,14.612,150.865
C05021=1107.809,342.853,415.694,-179.158,14.609,150.865
C05022=1107.801,342.485,415.744,-179.162,14.606,150.866
C05023=1107.795,342.237,415.777,-179.166,14.604,150.866
C05024=1107.789,341.989,415.811,-179.169,14.602,150.866
C05025=1107.784,341.741,415.845,-179.173,14.600,150.866
C05026=1107.778,341.494,415.878,-179.176,14.597,150.867
C05027=1107.772,341.246,415.911,-179.179,14.595,150.867
C05028=1107.766,340.998,415.944,-179.183,14.593,150.867
C05029=1107.761,340.750,415.977,-179.186,14.591,150.867
C05030=1107.755,340.503,416.012,-179.190,14.589,150.868
C05031=1107.749,340.255,416.045,-179.192,14.587,150.868
C05032=1107.744,340.008,416.078,-179.196,14.585,150.868
C05033=1107.739,339.760,416.111,-179.199,14.583,150.868
C05034=1107.733,339.512,416.144,-179.202,14.581,150.868
C05035=1107.727,339.264,416.177,-179.206,14.579,150.869
C05036=1107.721,339.016,416.211,-179.209,14.576,150.869
C05037=1107.716,338.769,416.244,-179.213,14.574,150.869
C05038=1107.710,338.521,416.277,-179.216,14.572,150.870
C05039=1107.704,338.273,416.310,-179.219,14.571,150.870
C05040=1107.699,338.025,416.343,-179.223,14.569,150.870
C05041=1107.693,337.777,416.377,-179.226,14.567,150.870
C05042=1107.687,337.530,416.409,-179.229,14.565,150.871
C05043=1107.682,337.282,416.442,-179.233,14.563,150.871
C05044=1107.676,337.035,416.476,-179.237,14.561,150.871
C05045=1107.670,336.787,416.508,-179.239,14.559,150.871
C05046=1107.664,336.539,416.542,-179.243,14.557,150.872
C05047=1107.659,336.291,416.575,-179.246,14.555,150.872
C05048=1107.652,336.044,416.608,-179.250,14.553,150.872
C05049=1107.647,335.795,416.641,-179.253,14.551,150.872
C05050=1107.642,335.548,416.673,-179.257,14.549,150.873
C05051=1107.636,335.300,416.706,-179.260,14.548,150.873
C05052=1107.630,335.052,416.740,-179.263,14.546,150.873
C05053=1107.625,334.804,416.773,-179.267,14.544,150.874
C05054=1107.619,334.557,416.806,-179.270,14.541,150.874
C05055=1107.613,334.308,416.838,-179.274,14.539,150.874
C05056=1107.608,334.061,416.871,-179.277,14.538,150.875
C05057=1107.602,333.813,416.904,-179.280,14.536,150.875
C05058=1107.597,333.566,416.937,-179.284,14.534,150.875
C05059=1107.591,333.317,416.969,-179.287,14.532,150.876
C05060=1107.586,333.070,417.002,-179.291,14.530,150.876
C05061=1107.579,332.823,417.035,-179.294,14.529,150.876
C05062=1107.574,332.574,417.068,-179.298,14.527,150.877
C05063=1107.568,332.326,417.101,-179.301,14.525,150.877
C05064=1107.562,332.079,417.134,-179.305,14.523,150.877
C05065=1107.557,331.831,417.165,-179.307,14.522,150.878
C05066=1107.551,331.583,417.199,-179.311,14.520,150.878
C05067=1107.545,331.336,417.231,-179.315,14.518,150.878
C05068=1107.540,331.087,417.264,-179.318,14.516,150.879
C05069=1107.533,330.839,417.297,-179.321,14.515,150.879
C05070=1107.528,330.592,417.329,-179.325,14.513,150.879
C05071=1107.519,330.217,417.378,-179.330,14.510,150.880
C05072=1107.510,329.843,417.427,-179.335,14.508,150.880
C05073=1107.502,329.469,417.476,-179.341,14.505,150.881
C05074=1107.493,329.094,417.525,-179.346,14.503,150.882
C05075=1107.487,328.847,417.559,-179.349,14.501,150.882
C05076=1107.482,328.599,417.590,-179.353,14.500,150.882
C05077=1107.476,328.351,417.623,-179.357,14.498,150.883
C05078=1107.470,328.103,417.655,-179.360,14.497,150.883
C05079=1107.464,327.855,417.689,-179.363,14.495,150.883
C05080=1107.459,327.608,417.720,-179.367,14.493,150.884
C05081=1107.453,327.360,417.752,-179.371,14.491,150.884
C05082=1107.447,327.112,417.786,-179.374,14.490,150.885
C05083=1107.442,326.864,417.817,-179.378,14.488,150.885
C05084=1107.436,326.617,417.850,-179.381,14.486,150.885
C05085=1107.430,326.368,417.882,-179.384,14.485,150.886
C05086=1107.424,326.120,417.915,-179.388,14.483,150.886
C05087=1107.419,325.873,417.947,-179.392,14.482,150.887
C05088=1107.413,325.625,417.979,-179.395,14.480,150.887
C05089=1107.407,325.377,418.011,-179.398,14.479,150.887
C05090=1107.402,325.129,418.043,-179.402,14.477,150.888
C05091=1107.396,324.881,418.076,-179.405,14.476,150.888
C05092=1107.390,324.634,418.108,-179.409,14.474,150.889
C05093=1107.384,324.385,418.140,-179.413,14.472,150.889
C05094=1107.378,324.137,418.172,-179.416,14.471,150.889
C05095=1107.373,323.890,418.205,-179.419,14.469,150.890
C05096=1107.367,323.642,418.237,-179.423,14.468,150.890
C05097=1107.361,323.394,418.269,-179.426,14.467,150.891
C05098=1107.356,323.146,418.300,-179.430,14.465,150.891
C05099=1107.350,322.898,418.332,-179.434,14.463,150.892
C05100=1107.345,322.650,418.364,-179.437,14.462,150.892
C05101=1107.339,322.402,418.397,-179.440,14.460,150.892
C05102=1107.334,322.155,418.429,-179.444,14.459,150.893
C05103=1107.328,321.907,418.461,-179.447,14.457,150.893
C05104=1107.322,321.658,418.493,-179.451,14.456,150.894
C05105=1107.316,321.411,418.525,-179.455,14.454,150.894
C05106=1107.310,321.163,418.557,-179.458,14.453,150.895
C05107=1107.305,320.915,418.589,-179.462,14.451,150.895
C05108=1107.299,320.667,418.621,-179.465,14.450,150.895
C05109=1107.294,320.419,418.652,-179.469,14.449,150.896
C05110=1107.288,320.171,418.685,-179.472,14.447,150.896
C05111=1107.283,319.923,418.716,-179.475,14.446,150.897
C05112=1107.277,319.675,418.748,-179.479,14.444,150.897
C05113=1107.272,319.428,418.780,-179.483,14.442,150.898
C05114=1107.266,319.180,418.812,-179.486,14.441,150.898
C05115=1107.260,318.932,418.844,-179.490,14.440,150.898
C05116=1107.254,318.684,418.876,-179.493,14.439,150.899
C05117=1107.249,318.436,418.907,-179.497,14.437,150.899
C05118=1107.244,318.188,418.938,-179.501,14.435,150.900
C05119=1107.238,317.940,418.971,-179.504,14.434,150.900
C05120=1107.232,317.692,419.002,-179.508,14.433,150.901
C05121=1107.226,317.444,419.034,-179.511,14.432,150.901
C05122=1107.221,317.197,419.066,-179.515,14.430,150.902
C05123=1107.212,316.815,419.115,-179.520,14.427,150.902
C05124=1107.204,316.434,419.163,-179.526,14.426,150.903
C05125=1107.196,316.053,419.211,-179.531,14.423,150.904
C05126=1107.187,315.671,419.260,-179.537,14.422,150.905
C05127=1107.181,315.423,419.292,-179.541,14.420,150.905
C05128=1107.175,315.175,419.324,-179.544,14.419,150.906
C05129=1107.170,314.927,419.355,-179.548,14.418,150.906
C05130=1107.164,314.679,419.386,-179.551,14.417,150.907
C05131=1107.158,314.431,419.418,-179.555,14.415,150.907
C05132=1107.152,314.183,419.450,-179.558,14.414,150.907
C05133=1107.147,313.935,419.481,-179.562,14.413,150.908
C05134=1107.141,313.688,419.512,-179.565,14.412,150.909
C05135=1107.135,313.440,419.544,-179.569,14.411,150.909
C05136=1107.130,313.191,419.575,-179.573,14.409,150.910
C05137=1107.123,312.944,419.606,-179.576,14.408,150.910
C05138=1107.118,312.696,419.638,-179.580,14.407,150.911
C05139=1107.112,312.447,419.669,-179.584,14.406,150.911
C05140=1107.106,312.200,419.700,-179.587,14.404,150.912
C05141=1107.101,311.952,419.731,-179.591,14.403,150.912
C05142=1107.095,311.704,419.763,-179.595,14.402,150.913
C05143=1107.089,311.456,419.794,-179.598,14.401,150.913
C05144=1107.083,311.208,419.826,-179.602,14.400,150.914
C05145=1107.077,310.960,419.856,-179.605,14.399,150.914
C05146=1107.072,310.712,419.888,-179.609,14.398,150.915
C05147=1107.066,310.463,419.919,-179.613,14.397,150.916
C05148=1107.060,310.216,419.950,-179.616,14.395,150.916
C05149=1107.055,309.968,419.981,-179.620,14.395,150.917
C05150=1107.048,309.720,420.012,-179.624,14.393,150.917
C05151=1107.043,309.472,420.043,-179.627,14.392,150.918
C05152=1107.038,309.225,420.075,-179.631,14.390,150.918
C05153=1107.031,308.976,420.106,-179.634,14.390,150.919
C05154=1107.026,308.729,420.137,-179.638,14.388,150.919
C05155=1107.020,308.481,420.168,-179.642,14.388,150.920
C05156=1107.015,308.233,420.199,-179.646,14.386,150.920
C05157=1107.008,307.985,420.230,-179.649,14.385,150.921
C05158=1107.003,307.737,420.261,-179.653,14.384,150.922
C05159=1106.998,307.489,420.291,-179.656,14.383,150.922
C05160=1106.992,307.241,420.324,-179.660,14.382,150.923
C05161=1106.986,306.992,420.354,-179.664,14.381,150.923
C05162=1106.981,306.745,420.385,-179.668,14.380,150.924
C05163=1106.976,306.496,420.416,-179.671,14.379,150.924
C05164=1106.969,306.249,420.447,-179.675,14.377,150.925
C05165=1106.963,306.001,420.478,-179.679,14.377,150.926
C05166=1106.958,305.753,420.508,-179.682,14.375,150.926
C05167=1106.952,305.505,420.539,-179.686,14.375,150.927
C05168=1106.947,305.257,420.570,-179.690,14.373,150.927
C05169=1106.940,305.009,420.601,-179.693,14.372,150.928
C05170=1106.935,304.761,420.632,-179.697,14.371,150.928
C05171=1106.929,304.513,420.663,-179.700,14.370,150.929
C05172=1106.924,304.265,420.693,-179.705,14.369,150.930
C05173=1106.919,304.017,420.724,-179.708,14.368,150.930
C05174=1106.913,303.769,420.755,-179.712,14.367,150.931
C05175=1106.905,303.390,420.802,-179.717,14.366,150.932
C05176=1106.896,303.012,420.849,-179.723,14.364,150.932
C05177=1106.887,302.633,420.896,-179.729,14.362,150.933
C05178=1106.878,302.254,420.943,-179.734,14.361,150.934
C05179=1106.872,302.006,420.973,-179.739,14.360,150.935
C05180=1106.867,301.758,421.004,-179.742,14.359,150.935
C05181=1106.862,301.510,421.034,-179.745,14.358,150.936
C05182=1106.856,301.262,421.066,-179.749,14.357,150.937
C05183=1106.850,301.014,421.096,-179.753,14.356,150.937
C05184=1106.844,300.765,421.126,-179.757,14.355,150.938
C05185=1106.839,300.517,421.157,-179.760,14.354,150.938
C05186=1106.834,300.269,421.187,-179.764,14.353,150.939
C05187=1106.828,300.022,421.217,-179.767,14.352,150.940
C05188=1106.823,299.773,421.248,-179.772,14.351,150.940
C05189=1106.817,299.526,421.279,-179.775,14.350,150.941
C05190=1106.811,299.278,421.309,-179.778,14.349,150.941
C05191=1106.806,299.030,421.340,-179.783,14.348,150.942
C05192=1106.800,298.782,421.370,-179.786,14.347,150.943
C05193=1106.795,298.533,421.400,-179.790,14.346,150.943
C05194=1106.789,298.286,421.430,-179.794,14.346,150.944
C05195=1106.784,298.037,421.461,-179.798,14.344,150.944
C05196=1106.778,297.790,421.492,-179.801,14.344,150.945
C05197=1106.772,297.542,421.522,-179.805,14.343,150.946
C05198=1106.767,297.293,421.552,-179.809,14.342,150.946
C05199=1106.760,297.045,421.582,-179.812,14.341,150.947
C05200=1106.754,296.797,421.613,-179.816,14.340,150.948
C05201=1106.749,296.549,421.643,-179.820,14.339,150.948
C05202=1106.743,296.301,421.673,-179.823,14.339,150.949
C05203=1106.738,296.053,421.704,-179.827,14.338,150.950
C05204=1106.732,295.805,421.734,-179.831,14.337,150.950
C05205=1106.727,295.556,421.764,-179.835,14.336,150.951
C05206=1106.721,295.308,421.794,-179.838,14.335,150.952
C05207=1106.715,295.061,421.824,-179.842,14.335,150.952
C05208=1106.710,294.812,421.854,-179.846,14.334,150.953
C05209=1106.704,294.564,421.884,-179.850,14.333,150.954
C05210=1106.698,294.317,421.915,-179.853,14.333,150.954
C05211=1106.692,294.068,421.944,-179.857,14.331,150.955
C05212=1106.687,293.820,421.975,-179.861,14.331,150.956
C05213=1106.681,293.572,422.004,-179.865,14.330,150.956
C05214=1106.675,293.324,422.035,-179.868,14.329,150.957
C05215=1106.670,293.076,422.064,-179.872,14.328,150.957
C05216=1106.664,292.828,422.095,-179.876,14.327,150.958
C05217=1106.658,292.579,422.124,-179.880,14.327,150.959
C05218=1106.653,292.332,422.155,-179.883,14.326,150.959
C05219=1106.647,292.083,422.184,-179.887,14.325,150.960
C05220=1106.641,291.835,422.215,-179.891,14.325,150.961
C05221=1106.636,291.587,422.244,-179.894,14.324,150.961
C05222=1106.630,291.339,422.274,-179.899,14.323,150.962
C05223=1106.624,291.091,422.304,-179.902,14.322,150.963
C05224=1106.618,290.843,422.334,-179.906,14.321,150.964
C05225=1106.612,290.595,422.364,-179.910,14.321,150.964
C05226=1106.607,290.347,422.393,-179.914,14.320,150.965
C05227=1106.599,289.982,422.437,-179.919,14.319,150.966
C05228=1106.590,289.617,422.481,-179.925,14.318,150.967
C05229=1106.582,289.252,422.524,-179.930,14.317,150.968
C05230=1106.574,288.888,422.568,-179.936,14.316,150.969
C05231=1106.568,288.640,422.598,-179.940,14.316,150.970
C05232=1106.562,288.391,422.628,-179.943,14.315,150.970
C05233=1106.557,288.143,422.658,-179.947,14.314,150.971
C05234=1106.551,287.895,422.687,-179.951,14.314,150.972
C05235=1106.545,287.647,422.717,-179.954,14.313,150.972
C05236=1106.539,287.399,422.747,-179.959,14.312,150.973
C05237=1106.534,287.150,422.776,-179.963,14.312,150.974
C05238=1106.528,286.902,422.806,-179.966,14.311,150.975
C05239=1106.522,286.654,422.835,-179.970,14.310,150.975
C05240=1106.517,286.406,422.865,-179.974,14.310,150.976
C05241=1106.511,286.158,422.894,-179.977,14.309,150.977
C05242=1106.505,285.910,422.924,-179.982,14.308,150.977
C05243=1106.500,285.661,422.953,-179.985,14.308,150.978
C05244=1106.494,285.413,422.983,-179.989,14.308,150.979
C05245=1106.489,285.165,423.012,-179.993,14.307,150.980
C05246=1106.482,284.916,423.041,-179.997,14.306,150.980
C05247=1106.477,284.669,423.071,180.000,14.305,150.981
C05248=1106.472,284.421,423.101,179.996,14.305,150.982
C05249=1106.465,284.173,423.130,179.992,14.304,150.982
C05250=1106.460,283.924,423.160,179.988,14.304,150.983
C05251=1106.454,283.676,423.189,179.985,14.303,150.984
C05252=1106.449,283.428,423.218,179.980,14.302,150.984
C05253=1106.443,283.180,423.248,179.977,14.302,150.985
C05254=1106.438,282.931,423.277,179.973,14.302,150.986
C05255=1106.431,282.683,423.306,179.969,14.301,150.987
C05256=1106.426,282.435,423.336,179.965,14.300,150.987
C05257=1106.420,282.187,423.364,179.962,14.300,150.988
C05258=1106.415,281.938,423.394,179.958,14.299,150.989
C05259=1106.409,281.690,423.423,179.953,14.298,150.990
C05260=1106.403,281.442,423.452,179.950,14.298,150.990
C05261=1106.398,281.194,423.482,179.946,14.297,150.991
C05262=1106.392,280.946,423.511,179.943,14.297,150.992
C05263=1106.387,280.698,423.540,179.938,14.296,150.992
C05264=1106.380,280.449,423.569,179.935,14.296,150.993
C05265=1106.375,280.201,423.599,179.931,14.296,150.994
C05266=1106.369,279.953,423.627,179.927,14.295,150.995
C05267=1106.364,279.704,423.656,179.923,14.294,150.995
C05268=1106.358,279.456,423.686,179.919,14.294,150.996
C05269=1106.352,279.208,423.715,179.916,14.294,150.997
C05270=1106.347,278.960,423.744,179.912,14.293,150.998
C05271=1106.341,278.711,423.773,179.908,14.292,150.998
C05272=1106.335,278.463,423.802,179.904,14.292,150.999
C05273=1106.329,278.216,423.830,179.901,14.291,151.000
C05274=1106.324,277.967,423.860,179.897,14.291,151.001
C05275=1106.318,277.719,423.888,179.892,14.290,151.001
C05276=1106.312,277.470,423.918,179.889,14.290,151.002
C05277=1106.307,277.223,423.947,179.885,14.290,151.003
C05278=1106.302,276.974,423.976,179.882,14.289,151.004
C05279=1106.293,276.619,424.016,179.876,14.289,151.005
C05280=1106.285,276.263,424.058,179.870,14.288,151.006
C05281=1106.277,275.908,424.100,179.865,14.287,151.007
C05282=1106.269,275.553,424.141,179.859,14.287,151.008
C05283=1106.263,275.304,424.170,179.855,14.286,151.009
C05284=1106.257,275.056,424.198,179.852,14.286,151.010
C05285=1106.252,274.807,424.227,179.848,14.286,151.010
C05286=1106.246,274.560,424.256,179.843,14.285,151.011
C05287=1106.240,274.311,424.284,179.840,14.285,151.012
C05288=1106.235,274.063,424.314,179.836,14.284,151.013
C05289=1106.229,273.815,424.342,179.833,14.284,151.013
C05290=1106.223,273.567,424.371,179.828,14.283,151.014
C05291=1106.217,273.318,424.399,179.824,14.283,151.015
C05292=1106.212,273.070,424.429,179.821,14.283,151.016
C05293=1106.206,272.821,424.457,179.817,14.282,151.017
C05294=1106.200,272.573,424.486,179.813,14.282,151.017
C05295=1106.195,272.325,424.514,179.809,14.281,151.018
C05296=1106.190,272.076,424.543,179.805,14.281,151.019
C05297=1106.184,271.829,424.572,179.802,14.281,151.020
C05298=1106.178,271.580,424.600,179.798,14.281,151.020
C05299=1106.172,271.332,424.629,179.794,14.280,151.021
C05300=1106.166,271.084,424.657,179.790,14.280,151.022
C05301=1106.160,270.835,424.685,179.786,14.279,151.023
C05302=1106.156,270.587,424.714,179.782,14.279,151.024
C05303=1106.150,270.338,424.743,179.778,14.279,151.024
C05304=1106.144,270.090,424.771,179.775,14.279,151.025
C05305=1106.138,269.842,424.799,179.770,14.278,151.026
C05306=1106.132,269.594,424.828,179.767,14.277,151.027
C05307=1106.127,269.345,424.856,179.763,14.277,151.028
C05308=1106.121,269.097,424.884,179.759,14.277,151.028
C05309=1106.115,268.849,424.912,179.755,14.277,151.029
C05310=1106.109,268.601,424.941,179.751,14.277,151.030
C05311=1106.104,268.352,424.969,179.747,14.276,151.031
C05312=1106.099,268.103,424.998,179.743,14.276,151.032
C05313=1106.093,267.855,425.026,179.739,14.276,151.032
C05314=1106.087,267.607,425.055,179.736,14.275,151.033
C05315=1106.081,267.358,425.084,179.732,14.275,151.034
C05316=1106.076,267.110,425.112,179.728,14.275,151.035
C05317=1106.070,266.862,425.140,179.724,14.274,151.036
C05318=1106.065,266.614,425.168,179.720,14.274,151.036
C05319=1106.059,266.365,425.196,179.716,14.274,151.037
C05320=1106.053,266.117,425.224,179.713,14.274,151.038
C05321=1106.047,265.868,425.252,179.709,14.274,151.039
C05322=1106.042,265.620,425.280,179.705,14.274,151.040
C05323=1106.037,265.372,425.308,179.701,14.273,151.040
C05324=1106.031,265.123,425.337,179.697,14.272,151.041
C05325=1106.025,264.875,425.365,179.693,14.272,151.042
C05326=1106.019,264.626,425.393,179.689,14.272,151.043
C05327=1106.014,264.378,425.421,179.686,14.272,151.044
C05328=1106.007,264.130,425.449,179.682,14.272,151.045
C05329=1106.002,263.882,425.477,179.678,14.272,151.045
C05330=1105.996,263.633,425.505,179.673,14.271,151.046
C05331=1105.988,263.281,425.545,179.668,14.271,151.047
C05332=1105.980,262.928,425.585,179.662,14.270,151.049
C05333=1105.972,262.575,425.624,179.657,14.270,151.050
C05334=1105.963,262.224,425.663,179.652,14.271,151.051
C05335=1105.957,261.975,425.692,179.647,14.270,151.052
C05336=1105.952,261.727,425.720,179.643,14.270,151.053
C05337=1105.946,261.478,425.748,179.640,14.269,151.053
C05338=1105.940,261.230,425.775,179.636,14.269,151.054
C05339=1105.934,260.981,425.803,179.632,14.269,151.055
C05340=1105.929,260.733,425.831,179.628,14.269,151.056
C05341=1105.923,260.484,425.859,179.624,14.269,151.057
C05342=1105.917,260.236,425.887,179.620,14.269,151.058
C05343=1105.912,259.988,425.915,179.616,14.269,151.059
C05344=1105.906,259.739,425.942,179.612,14.268,151.059
C05345=1105.900,259.491,425.970,179.608,14.268,151.060
C05346=1105.894,259.242,425.998,179.604,14.268,151.061
C05347=1105.889,258.994,426.026,179.601,14.268,151.062
C05348=1105.884,258.746,426.053,179.597,14.268,151.063
C05349=1105.877,258.497,426.081,179.593,14.268,151.064
C05350=1105.871,258.249,426.109,179.589,14.268,151.065
C05351=1105.866,258.000,426.136,179.585,14.268,151.065
C05352=1105.860,257.752,426.164,179.582,14.268,151.066
C05353=1105.854,257.504,426.192,179.577,14.267,151.067
C05354=1105.848,257.255,426.219,179.573,14.267,151.068
C05355=1105.843,257.007,426.247,179.569,14.267,151.069
C05356=1105.838,256.758,426.274,179.565,14.267,151.070
C05357=1105.831,256.510,426.302,179.561,14.267,151.070
C05358=1105.826,256.262,426.330,179.558,14.267,151.071
C05359=1105.821,256.013,426.357,179.554,14.267,151.072
C05360=1105.814,255.765,426.385,179.550,14.267,151.073
C05361=1105.809,255.516,426.412,179.546,14.267,151.074
C05362=1105.803,255.268,426.439,179.542,14.267,151.075
C05363=1105.798,255.020,426.466,179.538,14.267,151.075
C05364=1105.792,254.771,426.495,179.534,14.266,151.076
C05365=1105.786,254.523,426.521,179.530,14.266,151.077
C05366=1105.781,254.274,426.549,179.526,14.266,151.078
C05367=1105.774,254.025,426.576,179.522,14.266,151.079
C05368=1105.769,253.777,426.604,179.519,14.266,151.080
C05369=1105.763,253.529,426.631,179.515,14.266,151.081
C05370=1105.758,253.280,426.658,179.511,14.266,151.081
C05371=1105.752,253.032,426.687,179.507,14.266,151.082
C05372=1105.746,252.783,426.713,179.503,14.266,151.083
C05373=1105.741,252.535,426.741,179.499,14.266,151.084
C05374=1105.735,252.287,426.768,179.495,14.266,151.085
C05375=1105.730,252.037,426.795,179.492,14.266,151.086
C05376=1105.724,251.790,426.823,179.487,14.265,151.087
C05377=1105.719,251.541,426.850,179.483,14.265,151.088
C05378=1105.713,251.293,426.877,179.479,14.265,151.088
C05379=1105.708,251.045,426.905,179.476,14.265,151.089
C05380=1105.701,250.796,426.932,179.472,14.265,151.090
C05381=1105.696,250.547,426.959,179.468,14.265,151.091
C05382=1105.690,250.299,426.985,179.464,14.265,151.092
C05383=1105.682,249.944,427.025,179.459,14.265,151.093
C05384=1105.674,249.588,427.064,179.453,14.264,151.094
C05385=1105.666,249.233,427.102,179.447,14.264,151.095
C05386=1105.658,248.878,427.140,179.442,14.264,151.097
C05387=1105.652,248.629,427.168,179.438,14.264,151.098
C05388=1105.647,248.381,427.195,179.434,14.264,151.098
C05389=1105.642,248.132,427.222,179.430,14.264,151.099
C05390=1105.636,247.884,427.249,179.426,14.264,151.100
C05391=1105.630,247.635,427.276,179.422,14.264,151.101
C05392=1105.625,247.387,427.303,179.418,14.264,151.102
C05393=1105.619,247.138,427.330,179.414,14.264,151.103
C05394=1105.614,246.890,427.356,179.410,14.264,151.104
C05395=1105.608,246.641,427.384,179.407,14.264,151.105
C05396=1105.602,246.392,427.410,179.403,14.264,151.105
C05397=1105.596,246.144,427.437,179.399,14.264,151.106
C05398=1105.591,245.895,427.464,179.395,14.264,151.107
C05399=1105.585,245.647,427.492,179.391,14.264,151.108
C05400=1105.579,245.399,427.518,179.387,14.264,151.109
C05401=1105.574,245.151,427.545,179.383,14.264,151.110
C05402=1105.569,244.901,427.572,179.379,14.264,151.111
C05403=1105.563,244.653,427.598,179.375,14.264,151.112
C05404=1105.557,244.404,427.625,179.372,14.264,151.112
C05405=1105.551,244.156,427.652,179.368,14.264,151.113
C05406=1105.546,243.907,427.679,179.364,14.264,151.114
C05407=1105.540,243.659,427.706,179.360,14.264,151.115
C05408=1105.534,243.410,427.732,179.356,14.264,151.116
C05409=1105.529,243.162,427.759,179.352,14.264,151.117
C05410=1105.523,242.914,427.786,179.348,14.265,151.118
C05411=1105.517,242.665,427.812,179.344,14.265,151.119
C05412=1105.511,242.417,427.839,179.340,14.265,151.120
C05413=1105.507,242.168,427.866,179.336,14.265,151.120
C05414=1105.501,241.919,427.892,179.332,14.265,151.121
C05415=1105.495,241.671,427.919,179.329,14.265,151.122
C05416=1105.489,241.422,427.945,179.325,14.265,151.123
C05417=1105.484,241.174,427.972,179.321,14.265,151.124
C05418=1105.478,240.925,427.998,179.317,14.265,151.125
C05419=1105.472,240.677,428.025,179.313,14.265,151.126
C05420=1105.466,240.428,428.052,179.309,14.265,151.127
